(* Logix 5000 project; controller AdvManLab vendor 1 type 14 code 158 rev 28.12; software revision 28.01; part 3 of 13 *)
(* tags used below, declared in another part *)
   Cfg_Exists : BOOL;   // 1=Alarm configured to exist, 0=Does not exist, don't scan
   Cfg_ResetReqd : BOOL;   // 1=Latched Alarm, a Reset is required to clear this Alarm
   Cfg_AckReqd : BOOL;   // 1=Acknowledge required for this Alarm
   Cfg_AllowShelve : BOOL;   // 1=Allow Operator to Shelve this Alarm
   Cfg_AllowDisable : BOOL;   // 1=Allow Maintenance to Disable this Alarm
   Cfg_Severity : INT;   // Alarm Severity: 1..250=Low, 251..500=Medium, 501..750=High, 751..1000=Urgent
   Cfg_AlmMinOnT : DINT;   // Minimum time Alm output stays on (sec)
   PCfg_AllowExist : BOOL;   // 1=Alarm can be configured to exist, 0=other configs make alarm meaningless
   PCmd_Ack : BOOL;   // Program Command to Acknowledge alarm
   PCmd_Suppress : BOOL;   // Program Command to Suppress by Design (inhibits new alarm)
   PCmd_Unsuppress : BOOL;   // Program Command to Unsuppress (allows new alarm)
   PCmd_Unshelve : BOOL;   // Program Command to Unshelve (e.g., on shift change)
   OCmd_Ack : BOOL;   // Operator Command to Acknowledge alarm
   OCmd_Shelve : BOOL;   // Operator Command to Shelve Alarm (inhibits new alarm)
   OCmd_Unshelve : BOOL;   // Operator Command to Unshelve alarm (allows new alarm)
   Alm : ALIAS FOR Com_AE.0;   // Alarm output 1=In Alarm
   Ack : ALIAS FOR Com_AE.1;   // Alarm acknowledged status: 1=Ack rcvd
   Shelved : ALIAS FOR Com_AE.3;   // 1=Alarm has been Shelved by Operator (inhibits new alarm)
   Suppressed : ALIAS FOR Com_AE.6;   // 1=Alarm has been Suppressed by Program (inhibits new alarm)
   Disabled : ALIAS FOR Com_AE.9;   // 1=Alarm has been Disabled by Maintanance (inhibits new alarm)
   P_Alarm : BOOL;   // Unique Parameter Name for auto - discovery
   Wrk_Suppressed : BOOL;   // Internal Alarm Suppressed Status
   Com_AE : INT;   // Communication with HMI / Alarm/Event Server (see bit descriptions)
   PF525 : PF525_Faceplate_AOI;
   Running : BOOL;
(* P_Alarm, continued *)

ROUTINE Prescan   (* ladder *)
// Clear "lurking" Commands
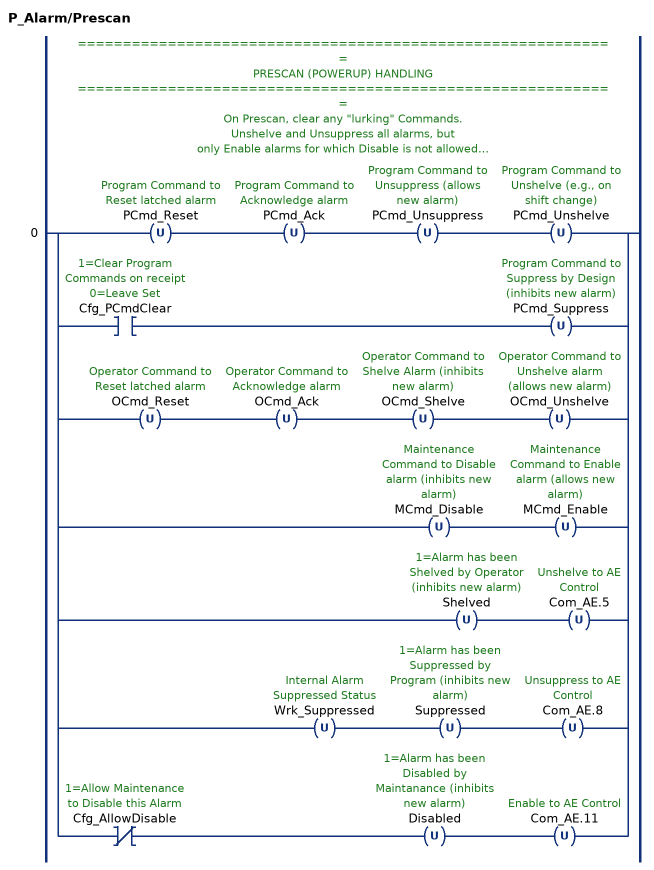
   // ============================================================
   // PRESCAN (POWERUP) HANDLING
   // ============================================================
   // On Prescan, clear any "lurking" Commands.
   // Unshelve and Unsuppress all alarms, but
   // only Enable alarms for which Disable is not allowed.
   // (Let Maintenance Disable persist through a power cycle...)
   // #####  V3.0-00  2013-06-30:  Added PCmd_Unshelve, AllowDisable, AllowShelve.  #####
   0: [OTU(PCmd_Reset) OTU(PCmd_Ack) OTU(PCmd_Unsuppress) OTU(PCmd_Unshelve) ,XIC(Cfg_PCmdClear) OTU(PCmd_Suppress) ,OTU(OCmd_Reset) OTU(OCmd_Ack) OTU(OCmd_Shelve) OTU(OCmd_Unshelve) ,OTU(MCmd_Disable) OTU(MCmd_Enable) ,OTU(Shelved) OTU(Com_AE.5) ,OTU(Wrk_Suppressed) OTU(Suppressed) OTU(Com_AE.8) ,XIO(Cfg_AllowDisable) OTU(Disabled) OTU(Com_AE.11) ];
END_ROUTINE
END_ADD_ON_INSTRUCTION

ADD_ON_INSTRUCTION P_Mode   (* revision 3.1 00 Release, vendor Rockwell Automation, ExecutePrescan, ExecuteEnableInFalse *)
// Mode
// Revision note:
// See Release Notes for Library version 3.1-xx for details. Containing objects must expose Maintenance
// Acquire / Release commands and new Sts_MAcqRcvd.
// Changed Val (enum) to SINT. Fixed parameter descriptions.
// Help:
// Copyright © Rockwell Automation, Inc.  All Rights Reserved.
// This instruction provides selection of Mode (owner) for a Device level
// object  (from highest priority to lowest):
// *  No Mode (no owner, EnableIn is false)
// *  Hand (typically tracks hardwired control of device)
// *  Maint (Maintenance) (taken out of normal service for maintenance)
// *  Ovrd (Override) (typically used for process overrides)
// *  Prog  (Program) (automated control, and default if Cfg_ProgNorm = 1)
// *  Oper (Operator (manual control, and default if Cfg_ProgNorm = 0)
// (Program and Operator have the same priority.)
// The current mode is shown with Status bits and also as the primary
// Value for the instruction: an enumeration "Val" as follows:
//   0 = No Mode,
//   1 = Hand,
//   2 = Maintenance,
//   3 = Override,
//   4 = Program (Locked),
//   5 = Operator (Locked),
//   6 = Program (Unlocked, Oper default),
//   7 = Operator (Unlocked, Prog default),
//   8 = Program (Unlocked, = default),
//   9 = Operator (Unlocked, = default).
// When EnableIn is false, all ownership acquire/release and lock/unlock
// Commands are processed "behind the scenes", but the Mode is shown
// as "No Mode" (no owner).  When EnableIn becomes true, the Mode
// takes into account the Commands received -- in other words, the Mode
// becomes the one that would have been in effect had the EnableIn
// False / No Mode condition never occurred.
VAR_INPUT
   Inp_Hand : BOOL; {visible}   // 1=Acquire Hand (typ. hardwired local) Mode, 0=Release Hand Mode
   Inp_Ovrd : BOOL; {visible}   // 1=Acquire Override (higher priority program logic) Mode, 0=Release Override Mode
   Cfg_PCmdClear : BOOL := 1;   // 1=Clear Program Command on receipt; 0=Use Level-based (maintained) PCmds
   Cfg_OvrdOverLock : BOOL := 1;   // 1=Override supersedes Prog/Oper Lock, 0=don't override Lock
   Cfg_ProgDefault : BOOL;   // Default Mode: 1=Program Mode if no requests; 0=Operator Mode if no requests
   PCmd_Acq : BOOL;   // Program Command to Acquire Ownership (Oper to Prog)
   PCmd_Rel : BOOL;   // Program Command to Release Ownership (Prog to Oper)
   PCmd_Lock : BOOL;   // Program Command to Lock Mode in Prog
   PCmd_Unlock : BOOL;   // Program Command to Unlock Mode
   MCmd_Acq : BOOL;   // Maintenance Command to Acquire Ownership (Oper/Prog/Ovrd to Maint)
   MCmd_Rel : BOOL;   // Maintenance Command to Release Ownership (Maint to Oper/Prog/Ovrd)
   OCmd_AcqLock : BOOL;   // Operator Command to Acquire (Prog to Oper) / Lock Ownership
   OCmd_UnlockRel : BOOL;   // Operator Command to Unlock / Release (Oper to Prog) Ownership
END_VAR
VAR_OUTPUT
   Val : SINT; {access Read Only}   // Mode enum: 0=No, 1=H, 2=M, 3=!, 4=P Lock, 5=O Lock, 6=P (O Def), 7=O (P Def), 8=P (= Def), 9=O (= Def)
   Sts_Hand : BOOL; {access Read Only, visible}   // 1=Mode is Hand (supersedes Maint, Ovrd, Prog, Oper)
   Sts_Maint : BOOL; {access Read Only, visible}   // 1=Mode is Maintenance (supersedes Ovrd, Prog, Oper)
   Sts_Ovrd : BOOL; {access Read Only, visible}   // 1=Mode is Override (supersedes Prog, Oper)
   Sts_Prog : BOOL; {access Read Only, visible}   // 1=Mode is Program
   Sts_Oper : BOOL := 1; {access Read Only, visible}   // 1=Mode is Operator
   Sts_ProgOperLock : BOOL; {access Read Only, visible}   // 1=Program or Operator has requested Mode Lock
   Sts_ProgOperSel : BOOL; {access Read Only}   // Prog/Oper selection 1=Program, 0=Operator
   Sts_NoMode : BOOL; {access Read Only}   // 1=Mode is No Mode (no owner, disabled or not scanned)
   Sts_MAcqRcvd : BOOL; {access Read Only}   // 1=Maintenance Acquire command received this scan
   Rdy_MAcq : BOOL; {access Read Only}   // 1=Ready for MCmd_Acq, enable button
   Rdy_MRel : BOOL; {access Read Only}   // 1=Ready for MCmd_Rel, enable button
   Rdy_OAcq : BOOL; {access Read Only}   // 1=Ready for OCmd_AcqLock, enable Acquire (to Oper) button
   Rdy_OLock : BOOL; {access Read Only}   // 1=Ready for OCmd_AcqLock, enable Oper Lock button
   Rdy_OUnlock : BOOL; {access Read Only}   // 1=Ready for OCmd_UnlockRel, enable Oper Unlock button
   Rdy_ORel : BOOL; {access Read Only}   // 1=Ready for OCmd_UnlockRel, enable Release (to Prog) button
   P_Mode : BOOL;   // Unique Parameter Name for auto - discovery
END_VAR
VAR
   Wrk_Locked : BOOL; {access None}   // 1=Program/Operator Mode selection is Locked
   Wrk_Prog : BOOL; {access None}   // Internal Program (1) / Operator (0) Mode selection
   Wrk_Maint : BOOL; {access None}   // Internal Maintenance Mode
   Inf_Lib : STRING_12 := 'RA-BAS'; {access Read Only}   // Display Library for Faceplate call-up
   Inf_Type : STRING_16 := 'P_Mode'; {access Read Only}   // Must contain AOI name, used for HMI and Information S/W
END_VAR

ROUTINE EnableInFalse   (* ladder *)
// Processes received Commands, but shows "NO mode" (no owner)
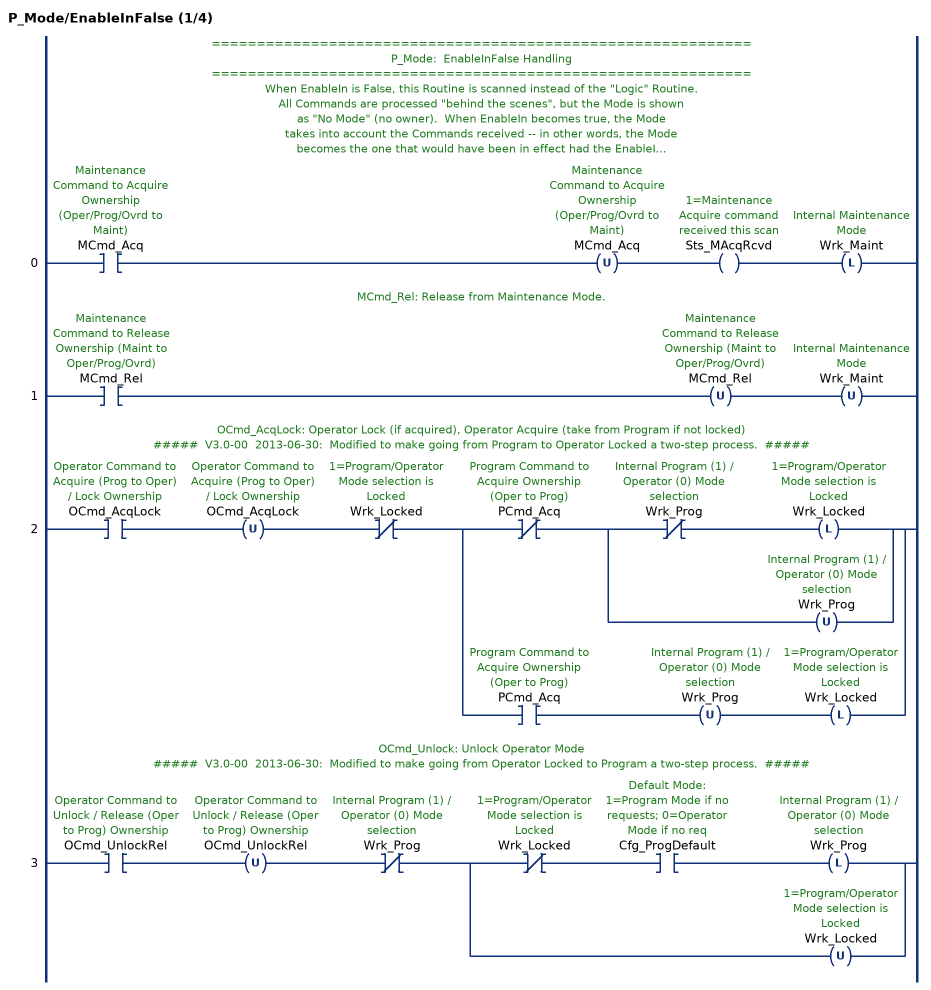
   // ============================================================
   // P_Mode:  EnableInFalse Handling
   // ============================================================
   // When EnableIn is False, this Routine is scanned instead of the "Logic" Routine.
   // All Commands are processed "behind the scenes", but the Mode is shown
   // as "No Mode" (no owner).  When EnableIn becomes true, the Mode
   // takes into account the Commands received -- in other words, the Mode
   // becomes the one that would have been in effect had the EnableIn
   // False / No Mode condition never occurred.
   // ============================================================
   // COMMAND HANDLING
   // ============================================================
   // NOTE:  These rungs MUST be in the order given to meet the following
   // multiple-actions-at-the-same-time scenarios:
   // * Maintenance Release beats Maintenance Acquire
   // * Program Release beats Program Acquire
   // * Program Unlock beats Program Lock
   // * Operator Unlock beats Operator Acquire and Lock (results in Oper Unlocked)
   // * Operator Acquire/Lock must come after Program Unlock
   // * Program Acquire must come after Operator Unlock
   // ===========================================================
   // MCmd_Acq: Acquire for Maintenance Mode, and blink the status
   // that indicates a Maintenance Acquire command was received.
   // #####  V3.1-00  2014-06-30:  Added Sts_MAcqRcvd  #####
   0: XIC(MCmd_Acq)OTU(MCmd_Acq)OTE(Sts_MAcqRcvd)OTL(Wrk_Maint);
   // MCmd_Rel: Release from Maintenance Mode.
   1: XIC(MCmd_Rel)OTU(MCmd_Rel)OTU(Wrk_Maint);
   // OCmd_AcqLock: Operator Lock (if acquired), Operator Acquire (take from Program if not locked)
   // #####  V3.0-00  2013-06-30:  Modified to make going from Program to Operator Locked a two-step process.  #####
   2: XIC(OCmd_AcqLock)OTU(OCmd_AcqLock)XIO(Wrk_Locked)[XIO(PCmd_Acq) [XIO(Wrk_Prog) OTL(Wrk_Locked) ,OTU(Wrk_Prog) ] ,XIC(PCmd_Acq) OTU(Wrk_Prog) OTL(Wrk_Locked) ];
   // OCmd_Unlock: Unlock Operator Mode
   // #####  V3.0-00  2013-06-30:  Modified to make going from Operator Locked to Program a two-step process.  #####
   3: XIC(OCmd_UnlockRel)OTU(OCmd_UnlockRel)XIO(Wrk_Prog)[XIO(Wrk_Locked) XIC(Cfg_ProgDefault) OTL(Wrk_Prog) ,OTU(Wrk_Locked) ];
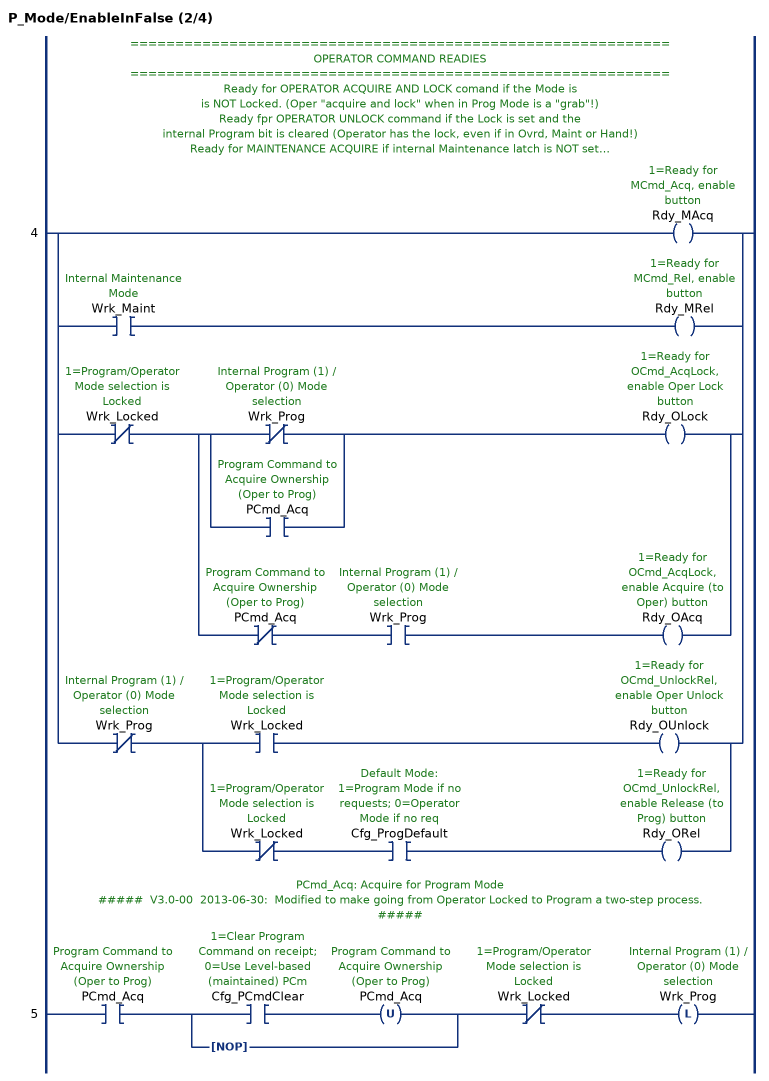
   // ============================================================
   // OPERATOR COMMAND READIES
   // ============================================================
   // Ready for OPERATOR ACQUIRE AND LOCK comand if the Mode is
   //  is NOT Locked. (Oper "acquire and lock" when in Prog Mode is a "grab"!)
   // Ready fpr OPERATOR UNLOCK command if the Lock is set and the
   // internal Program bit is cleared (Operator has the lock, even if in Ovrd, Maint or Hand!)
   // Ready for MAINTENANCE ACQUIRE if internal Maintenance latch is NOT set.
   // But we need to display Ready even if latch IS set so that Sts_MAcqRcvd
   // can blink to reset an external Maintenance expiration timer!!!
   // Ready for MAINTENANCE RELEASE if internal Maintenance latch IS set.
   // #####  V3.0-00  2013-06-30:  Modified Rdy_Unlock for two-step Operator Locked to Program process.  #####
   // #####  V3.1-00  2014-06-30:  Added Sts_MAcqRcvd  #####
   4: [OTE(Rdy_MAcq) ,XIC(Wrk_Maint) OTE(Rdy_MRel) ,XIO(Wrk_Locked) [[XIO(Wrk_Prog) ,XIC(PCmd_Acq) ] OTE(Rdy_OLock) ,XIO(PCmd_Acq) XIC(Wrk_Prog) OTE(Rdy_OAcq) ] ,XIO(Wrk_Prog) [XIC(Wrk_Locked) OTE(Rdy_OUnlock) ,XIO(Wrk_Locked) XIC(Cfg_ProgDefault) OTE(Rdy_ORel) ] ];
   // PCmd_Acq: Acquire for Program Mode
   // #####  V3.0-00  2013-06-30:  Modified to make going from Operator Locked to Program a two-step process.  #####
   5: XIC(PCmd_Acq)[XIC(Cfg_PCmdClear) OTU(PCmd_Acq) ,NOP() ]XIO(Wrk_Locked)OTL(Wrk_Prog);
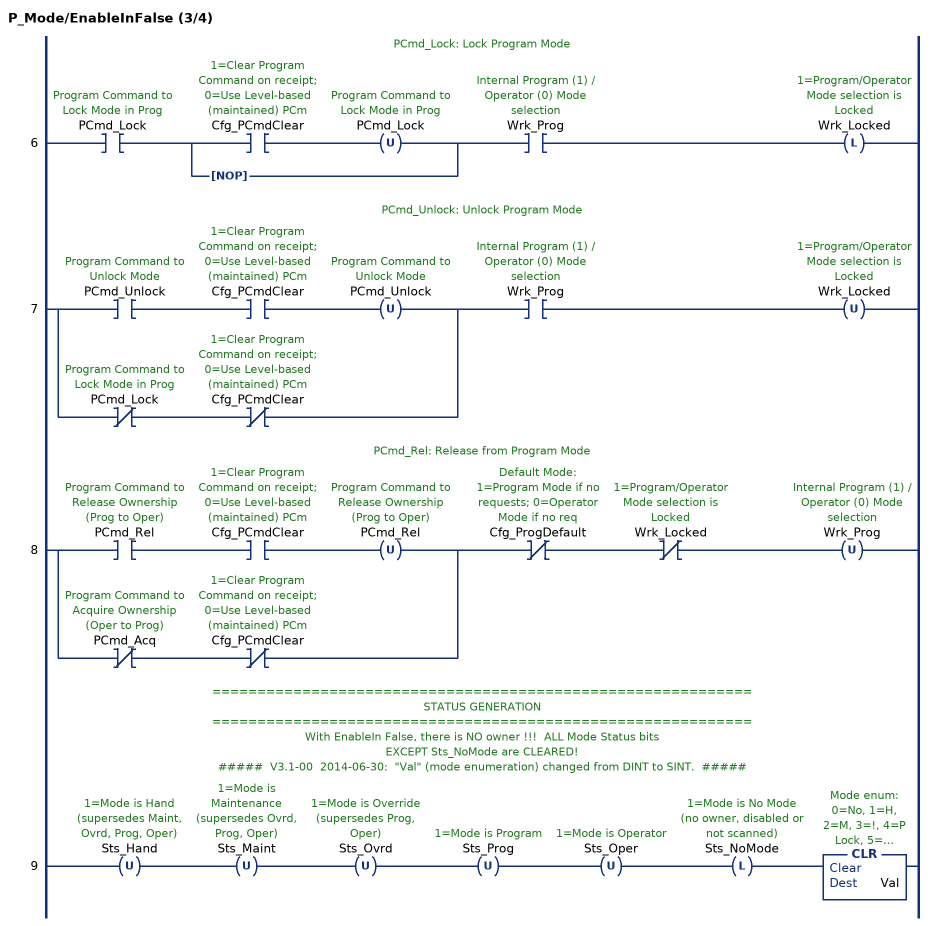
   // PCmd_Lock: Lock Program Mode
   6: XIC(PCmd_Lock)[XIC(Cfg_PCmdClear) OTU(PCmd_Lock) ,NOP() ]XIC(Wrk_Prog)OTL(Wrk_Locked);
   // PCmd_Unlock: Unlock Program Mode
   7: [XIC(PCmd_Unlock) XIC(Cfg_PCmdClear) OTU(PCmd_Unlock) ,XIO(PCmd_Lock) XIO(Cfg_PCmdClear) ]XIC(Wrk_Prog)OTU(Wrk_Locked);
   // PCmd_Rel: Release from Program Mode
   8: [XIC(PCmd_Rel) XIC(Cfg_PCmdClear) OTU(PCmd_Rel) ,XIO(PCmd_Acq) XIO(Cfg_PCmdClear) ]XIO(Cfg_ProgDefault)XIO(Wrk_Locked)OTU(Wrk_Prog);
   // ============================================================
   // STATUS GENERATION
   // ============================================================
   // With EnableIn False, there is NO owner !!!  ALL Mode Status bits
   // EXCEPT Sts_NoMode are CLEARED!
   // #####  V3.1-00  2014-06-30:  "Val" (mode enumeration) changed from DINT to SINT.  #####
   9: OTU(Sts_Hand)OTU(Sts_Maint)OTU(Sts_Ovrd)OTU(Sts_Prog)OTU(Sts_Oper)OTL(Sts_NoMode)CLR(Val);
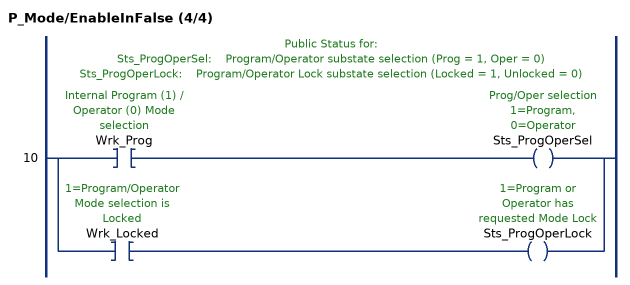
   // Public Status for:
   // Sts_ProgOperSel:    Program/Operator substate selection (Prog = 1, Oper = 0)
   // Sts_ProgOperLock:    Program/Operator Lock substate selection (Locked = 1, Unlocked = 0)
   10: [XIC(Wrk_Prog) OTE(Sts_ProgOperSel) ,XIC(Wrk_Locked) OTE(Sts_ProgOperLock) ];
END_ROUTINE

ROUTINE Logic   (* ladder *)
// Selects Modes (Hand, Maint, Ovrd, Oper, Prog) based on Inputs and Commands
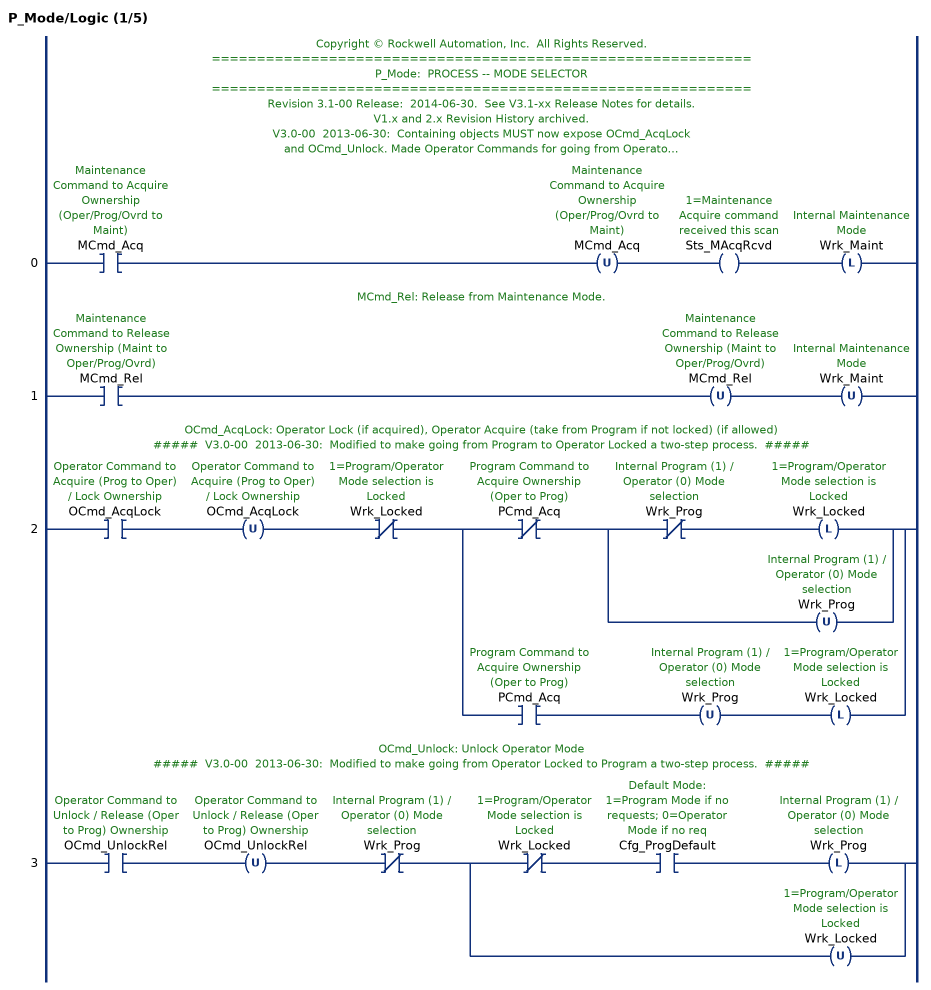
   // Copyright © Rockwell Automation, Inc.  All Rights Reserved.
   // ============================================================
   // P_Mode:  PROCESS -- MODE SELECTOR
   // ============================================================
   // Revision 3.1-00 Release:  2014-06-30.  See V3.1-xx Release Notes for details.
   // V1.x and 2.x Revision History archived.
   // V3.0-00  2013-06-30:  Containing objects MUST now expose OCmd_AcqLock
   // and OCmd_Unlock. Made Operator Commands for going from Operator
   // Locked to Program (unlocked) and Program (unlocked) to Operator
   // Lock two-step processes.  Added Inf_Lib, Inf_Type.
   // V3.1-00  2014-06-30: Containing objects must expose Maintenance
   // Acquire / Release commands and new Sts_MAcqRcvd.
   // Changed Val (enum) to SINT. Fixed parameter descriptions.
   // ============================================================
   // This instruction provides selection of Mode (owner) for a Device level
   // object  (from highest priority to lowest):
   // * NO Mode (EnableIn is false)
   // *  Hand (typically tracks hardwired control of device)
   // *  Maint (Maintenance) (taken out of normal service for maintenance)
   // *  Ovrd (Override) (typically used for process overrides)
   // *  Prog  (Program) (automated control, and default if Cfg_ProgNorm = 1)
   // *  Oper (Operator (manual control, and default if Cfg_ProgNorm = 0)
   // The current mode is shown with Status bits and also as the
   // primary Value for the instruction: an enumeration as follows:
   // 0 = No Mode, 1 = Hand, 2 = Maintenance, 3 = Override,
   // 4 = Program (Locked), 5 = Operator (Locked),
   // 6 = Program (Unlocked, Oper default), 7 = Operator (Unlocked, Prog default),
   // 8 = Program (Unlocked, Prog default), 9 = Operator (Unlocked, Oper default).
   // ============================================================
   // COMMAND HANDLING
   // ============================================================
   // NOTE:  These rungs MUST be in the order given to meet the following
   // multiple-actions-at-the-same-time scenarios:
   // * Maintenance Release beats Maintenance Acquire
   // * Program Release beats Program Acquire
   // * Program Unlock beats Program Lock
   // * Operator Unlock beats Operator Acquire / Lock (results in Oper Unlocked)
   // * Program Acquire must come after Operator Unlock
   // If Cfg_ProgDefault = 1, the Mode defaults to Program
   // (instead of Operator) if all other Modes release their requests.
   // ============================================================
   // MCmd_Acq: Acquire for Maintenance Mode, and blink the status
   // that indicates a Maintenance Acquire command was received.
   // #####  V3.1-00  2014-06-30:  Added Sts_MAcqRcvd  #####
   0: XIC(MCmd_Acq)OTU(MCmd_Acq)OTE(Sts_MAcqRcvd)OTL(Wrk_Maint);
   // MCmd_Rel: Release from Maintenance Mode.
   1: XIC(MCmd_Rel)OTU(MCmd_Rel)OTU(Wrk_Maint);
   // OCmd_AcqLock: Operator Lock (if acquired), Operator Acquire (take from Program if not locked) (if allowed)
   // #####  V3.0-00  2013-06-30:  Modified to make going from Program to Operator Locked a two-step process.  #####
   2: XIC(OCmd_AcqLock)OTU(OCmd_AcqLock)XIO(Wrk_Locked)[XIO(PCmd_Acq) [XIO(Wrk_Prog) OTL(Wrk_Locked) ,OTU(Wrk_Prog) ] ,XIC(PCmd_Acq) OTU(Wrk_Prog) OTL(Wrk_Locked) ];
   // OCmd_Unlock: Unlock Operator Mode
   // #####  V3.0-00  2013-06-30:  Modified to make going from Operator Locked to Program a two-step process.  #####
   3: XIC(OCmd_UnlockRel)OTU(OCmd_UnlockRel)XIO(Wrk_Prog)[XIO(Wrk_Locked) XIC(Cfg_ProgDefault) OTL(Wrk_Prog) ,OTU(Wrk_Locked) ];
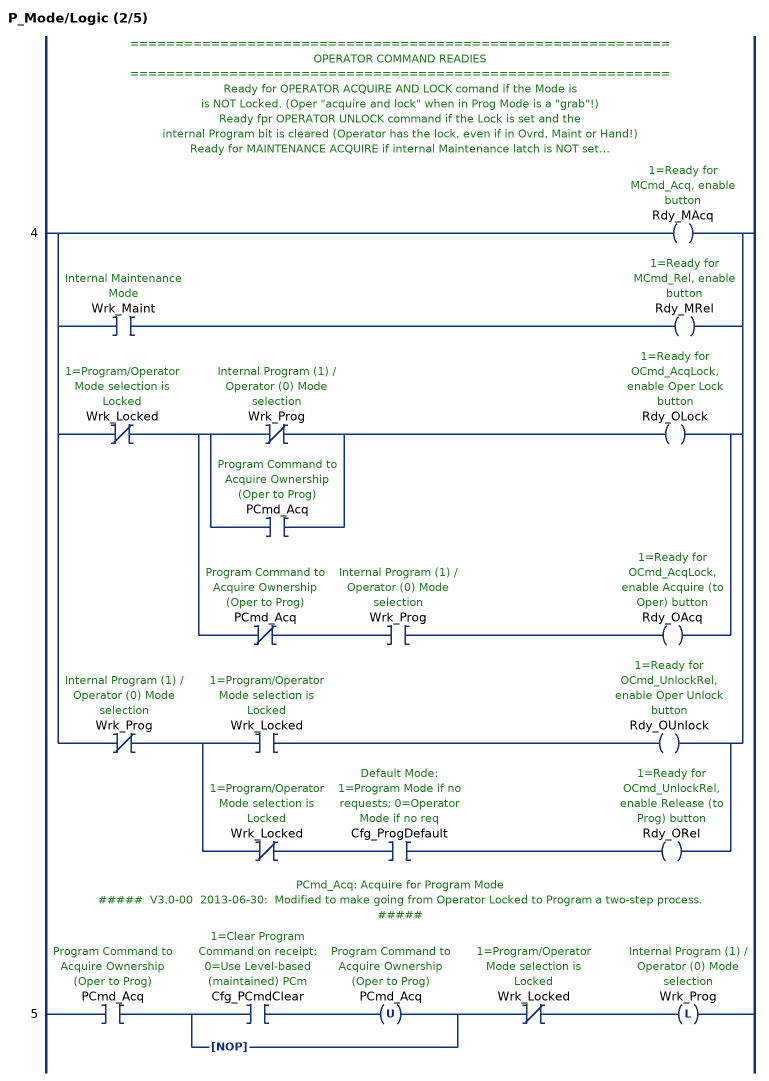
   // ============================================================
   // OPERATOR COMMAND READIES
   // ============================================================
   // Ready for OPERATOR ACQUIRE AND LOCK comand if the Mode is
   //  is NOT Locked. (Oper "acquire and lock" when in Prog Mode is a "grab"!)
   // Ready fpr OPERATOR UNLOCK command if the Lock is set and the
   // internal Program bit is cleared (Operator has the lock, even if in Ovrd, Maint or Hand!)
   // Ready for MAINTENANCE ACQUIRE if internal Maintenance latch is NOT set.
   // But we need to display Ready even if latch IS set so that Sts_MAcqRcvd
   // can blink to reset an external Maintenance expiration timer!!!
   // Ready for MAINTENANCE RELEASE if internal Maintenance latch IS set.
   // #####  V3.0-00  2013-06-30:  Modified Rdy_Unlock for two-step Operator Locked to Program process.  #####
   // #####  V3.1-00  2014-06-30:  Added Sts_MAcqRcvd  #####
   4: [OTE(Rdy_MAcq) ,XIC(Wrk_Maint) OTE(Rdy_MRel) ,XIO(Wrk_Locked) [[XIO(Wrk_Prog) ,XIC(PCmd_Acq) ] OTE(Rdy_OLock) ,XIO(PCmd_Acq) XIC(Wrk_Prog) OTE(Rdy_OAcq) ] ,XIO(Wrk_Prog) [XIC(Wrk_Locked) OTE(Rdy_OUnlock) ,XIO(Wrk_Locked) XIC(Cfg_ProgDefault) OTE(Rdy_ORel) ] ];
   // PCmd_Acq: Acquire for Program Mode
   // #####  V3.0-00  2013-06-30:  Modified to make going from Operator Locked to Program a two-step process.  #####
   5: XIC(PCmd_Acq)[XIC(Cfg_PCmdClear) OTU(PCmd_Acq) ,NOP() ]XIO(Wrk_Locked)OTL(Wrk_Prog);
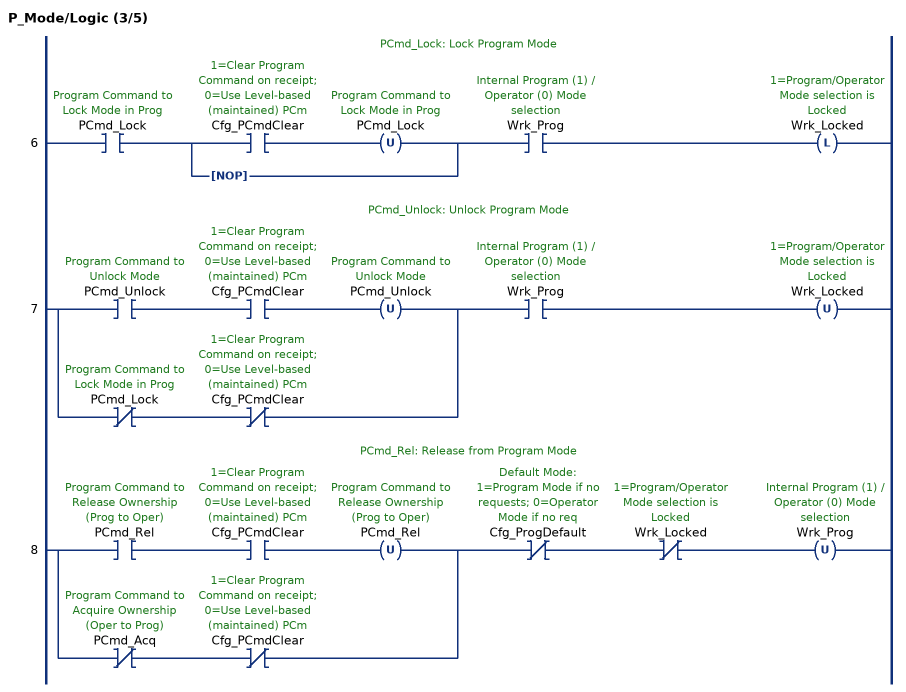
   // PCmd_Lock: Lock Program Mode
   6: XIC(PCmd_Lock)[XIC(Cfg_PCmdClear) OTU(PCmd_Lock) ,NOP() ]XIC(Wrk_Prog)OTL(Wrk_Locked);
   // PCmd_Unlock: Unlock Program Mode
   7: [XIC(PCmd_Unlock) XIC(Cfg_PCmdClear) OTU(PCmd_Unlock) ,XIO(PCmd_Lock) XIO(Cfg_PCmdClear) ]XIC(Wrk_Prog)OTU(Wrk_Locked);
   // PCmd_Rel: Release from Program Mode
   8: [XIC(PCmd_Rel) XIC(Cfg_PCmdClear) OTU(PCmd_Rel) ,XIO(PCmd_Acq) XIO(Cfg_PCmdClear) ]XIO(Cfg_ProgDefault)XIO(Wrk_Locked)OTU(Wrk_Prog);
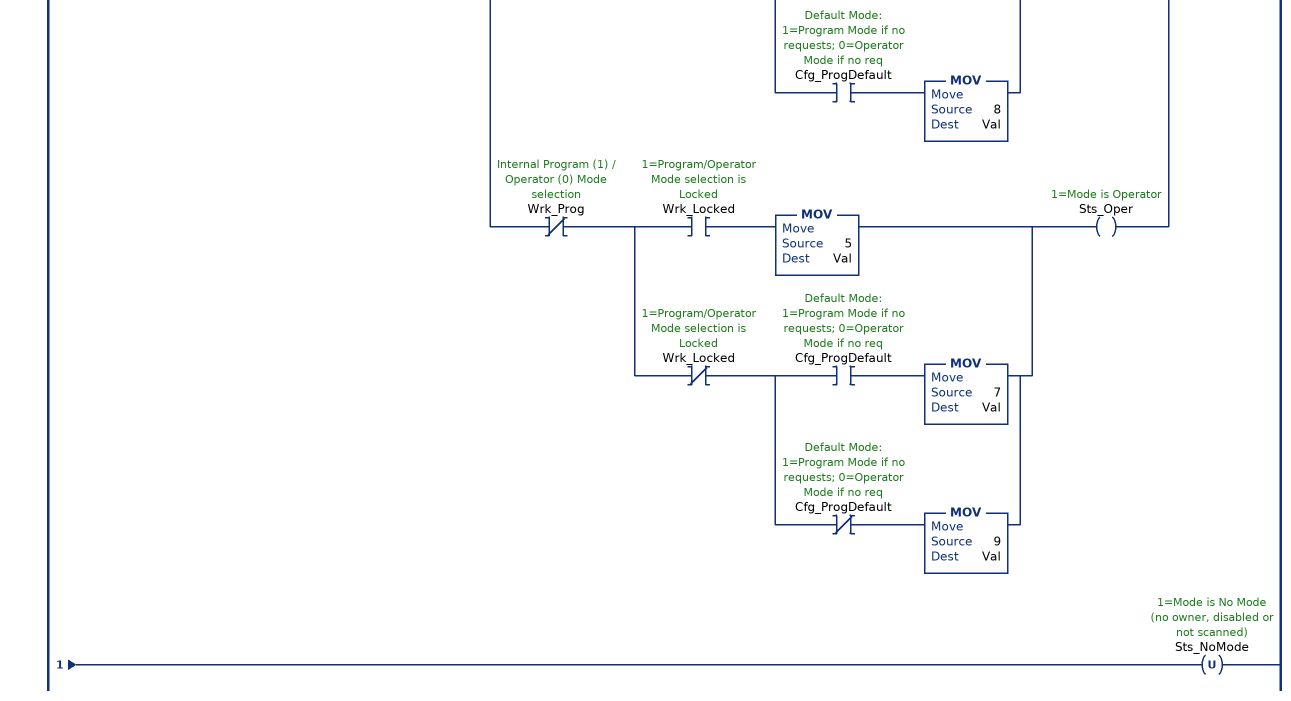
   // ============================================================
   // STATUS GENERATION
   // ============================================================
   // This rung determines the Mode based on the states of the inputs and internal working bits.
   // The logic here does the vast mahority of the implementation of the Mode selection rules.
   // Between the internal working bits used above and the rules implemented here,
   // outside objects cannot manipulate the state of this object by setting/clearing its Status bits.
   // Public Status is generated for:
   // *  Hand Mode
   // *  Maintenance Mode
   // *  Override Mode
   // *  Program Mode
   // *  Operator Mode
   // *  No Mode (none of the above)
   // #####  V3.1-00  2014-06-30:  "Val" (mode enumeration) changed from DINT to SINT.  #####
   9: [XIC(Inp_Hand) OTE(Sts_Hand) MOV(1,Val) ,XIO(Inp_Hand) [XIC(Wrk_Maint) OTE(Sts_Maint) MOV(2,Val) ,XIO(Wrk_Maint) [XIC(Inp_Ovrd) [XIO(Wrk_Locked) ,XIC(Cfg_OvrdOverLock) ,XIC(Sts_Ovrd) ] OTE(Sts_Ovrd) MOV(3,Val) ,XIO(Sts_Ovrd) [XIC(Wrk_Prog) [XIC(Wrk_Locked) MOV(4,Val) ,XIO(Wrk_Locked) [XIO(Cfg_ProgDefault) MOV(6,Val) ,XIC(Cfg_ProgDefault) MOV(8,Val) ] ] OTE(Sts_Prog) ,XIO(Wrk_Prog) [XIC(Wrk_Locked) MOV(5,Val) ,XIO(Wrk_Locked) [XIC(Cfg_ProgDefault) MOV(7,Val) ,XIO(Cfg_ProgDefault) MOV(9,Val) ] ] OTE(Sts_Oper) ] ] ] ]OTU(Sts_NoMode);
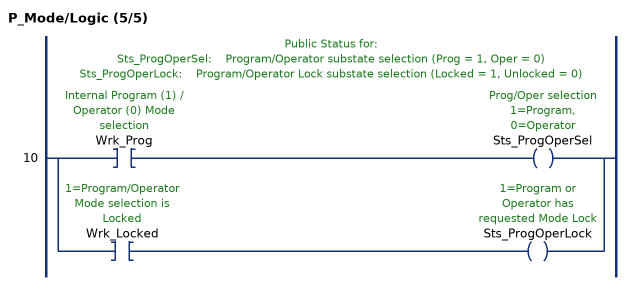
   // Public Status for:
   // Sts_ProgOperSel:    Program/Operator substate selection (Prog = 1, Oper = 0)
   // Sts_ProgOperLock:    Program/Operator Lock substate selection (Locked = 1, Unlocked = 0)
   10: [XIC(Wrk_Prog) OTE(Sts_ProgOperSel) ,XIC(Wrk_Locked) OTE(Sts_ProgOperLock) ];
END_ROUTINE

ROUTINE Prescan   (* ladder *)
// Clear "lurking" Commands
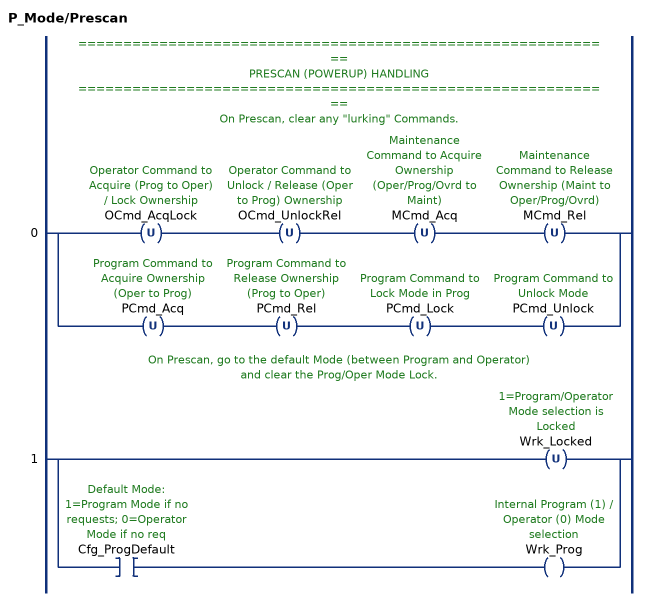
   // ============================================================
   // PRESCAN (POWERUP) HANDLING
   // ============================================================
   // On Prescan, clear any "lurking" Commands.
   0: [OTU(OCmd_AcqLock) OTU(OCmd_UnlockRel) OTU(MCmd_Acq) OTU(MCmd_Rel) ,OTU(PCmd_Acq) OTU(PCmd_Rel) OTU(PCmd_Lock) OTU(PCmd_Unlock) ];
   // On Prescan, go to the default Mode (between Program and Operator)
   // and clear the Prog/Oper Mode Lock.
   1: [OTU(Wrk_Locked) ,XIC(Cfg_ProgDefault) OTE(Wrk_Prog) ];
END_ROUTINE
END_ADD_ON_INSTRUCTION

ADD_ON_INSTRUCTION P_PF52x   (* revision 3.1 00 Release, vendor Rockwell Automation, ExecutePrescan, ExecuteEnableInFalse *)
// PowerFlex 523 / 525
// Variable Frequency Drive
// Revision note:
// See V3.1-xx Release Notes for Library for details. New instruction for PlantPAx Library 3.1.
// Help:
// Copyright © Rockwell Automation, Inc.  All Rights Reserved.
// This Instruction controls and monitors a PowerFlex 523 Variable-Frequency Drive with
// optional EtherNet/IP Interface, or a PowerFlex 525 Variable-Frequency Drive with
// embedded or optional add-on EtherNet/IP Interface.
// This instruction provides:
// *  Starting, stopping, jogging of drive, setting speed reference and direction
// *  Monitoring of run feedback, display of actual drive status, including accel, decel, direction, speed
// *  Detection of Failure to Start, Failure to Stop, Drive Fault
// *  Monitoring of Permissive conditions to allow starting
// *  Monitoring of Interlock conditions to stop / prevent starting
// *  Simulation, providing feedback of a working drive while disabling outputs
// *  Monitoring of I/O communication faults
// *  Alarms for Fail to Start, Fail to Stop, Interlock Trip, Drive Fault, I/O Fault
// *  Option to automatically reset faults and alarms when operator commands
//     motor to start or stop
// * Supports HMI "breadcrumbs" for Alarm Inhibited, Bad Configuration,
//     Not Ready, Maintenance Bypass Active
// * "Available" status for use by automation logic to know whether motor
//     can be controlled by other objects.
// See Rockwell Automation Publication 520COM-UM001_ for information on
// the PowerFlex 525 embedded EtherNet/IP interface.
// See Rockwell Automation Publication 520COM-UM003_ for information on
// the PowerFlex 525 add-on EtherNet/IP interface (dual-port).
// See Rockwell Automation Publication 520-UM001_ for information on the
// PowerFlex 523 and 525 drive parameters and programming
// Modes are provided by a P_Mode AOI instance.
// Alarms are provided by P_Alarm AOI instances.
// Modes of operation: Operator, Program, Override, Maintenance, Hand
// REQUIRED DRIVE CONFIGURATION
// Be certain to set up the drive Datalinks as follows!
// 'User Choice' Datalinks are not used by this AOI and
// may be left unused or set up for your application.
// INPUT ASSEMBLY:
// Drive Status (standard)
// Output Frequency (standard)
// 1. Fault 1 Code (Par 007)
// 2. Output Current (Par 003)
// 3. Output Power (Par 017)
// 4. User choice
// OUTPUT ASSEMBLY:
// Drive Logic Comnmand (standard)
// Frequency Command (Speed Reference) (standard)
// All 4 output datalinks are user choice.
VAR_IN_OUT
   Inp : P_PF52x_Inp; {required}   // Common part of PF523 / PF525 Input Assembly
   Out : P_PF52x_Out; {required}   // Common part of PF523 / PF525 Output Assembly
   Ref_FaultCodeList : P_DescList[1]; {required}   // Tag containing List of Fault Codes (DINT) and their Descriptions (STRING)
END_VAR
VAR_INPUT
   Inp_FwdPermOK : BOOL := 1; {visible}   // 1=Permissives OK, drive can start Forward
   Inp_FwdNBPermOK : BOOL := 1; {visible}   // 1=Non-Bypassable Permissives OK, drive can start Forward
   Inp_RevPermOK : BOOL := 1; {visible}   // 1=Permissives OK, drive can start Reverse
   Inp_RevNBPermOK : BOOL := 1; {visible}   // 1=Non-Bypassable Permissives OK, motor can start Reverse
   Inp_IntlkOK : BOOL := 1; {visible}   // 1=Interlocks OK, drive can start/run
   Inp_NBIntlkOK : BOOL := 1; {visible}   // 1=Non-Bypassable Interlocks OK, drive can start/run
   Inp_IOFault : BOOL;   // Input Communication Status 0=OK, 1=fail
   Inp_Sim : BOOL;   // 1=Simulate working drive; 0=Start/Stop/ Monitor actual drive
   Inp_Hand : BOOL; {visible}   // 1=Acquire Hand (typ. hardwired local) Mode, 0=Release Hand Mode
   Inp_Ovrd : ALIAS FOR Mode.Inp_Ovrd; {visible}
   Inp_OvrdCmd : SINT; {visible}   // Override Mode Command: 0=None, 1=Stop, 2=Start Fwd 3=Start Rev
   Inp_OvrdSpeed : REAL;   // Value to set Speed Reference in Override Mode (SpeedRef EU)
   Inp_Reset : BOOL; {visible}   // 1=Reset drive fault conditions and latched Alarms
   Cfg_HasReverse : BOOL;   // 1=Drive can be run reverse, 0=Forward only
   Cfg_HasJog : BOOL;   // 1=Drive Jog Command enabled/visible, 0=Drive Jog Command not allowed
   Cfg_AllowLocal : BOOL;   // 1=Allow Local Start/Stop without alarm, 0=Start/Stop from HMI/prog only
   Cfg_HasFwdPermObj : BOOL;   // 1=Tells HMI a P_Perm is connected to Inp_FwdPerm
   Cfg_HasRevPermObj : BOOL;   // 1=Tells HMI a P_Perm is connected to Inp_RevPerm
   Cfg_HasIntlkObj : BOOL;   // 1=Tells HMI a P_Intlk is connected to Inp_Intlk
   Cfg_HasResInhObj : BOOL;   // 1=Tells HMI a P_ResInh Restart Inhibit is connected
   Cfg_HasRunTimeObj : BOOL;   // 1=Tells HMI a P_RunTime is connected
   Cfg_SetTrack : BOOL := 1;   // 1=PSets track OSets in Oper, OSets track PSets in Prog, 0=no tracking
   Cfg_SetTrackOvrdHand : BOOL;   // 1=Prog/Oper Settings track Override/Hand speed reference
   Cfg_PCmdClear : ALIAS FOR Mode.Cfg_PCmdClear;
   Cfg_ProgDefault : ALIAS FOR Mode.Cfg_ProgDefault;
   Cfg_OperStopPrio : BOOL;   // 1=OCmd_Stop has priority, accepted any time, 0=OCmd_Stop only in Oper, Maint Mode.
   Cfg_OCmdResets : BOOL;   // 1=New Oper drive cmd. resets fault, 0=reset req'd to clear fault
   Cfg_OvrdPermIntlk : BOOL;   // 1=Override ignores Bypassable Perm/ Intlk; 0=always use Perm/Intlk
   Cfg_ShedOnFailToStart : BOOL := 1;   // 1=Stop Motor and Alarm on Fail to Start; 0=Alarm only on Fail to Start
   Cfg_ShedOnIOFault : BOOL := 1;   // 1=Stop Motor and Alarm on I/O Fault; 0=Alarm only on I/O Fault
   Cfg_SimScaleEU : BOOL;   // 1=In simulation, scale Speed Ref EU to Speed Fdbk EU
   Cfg_SimScaleRaw : BOOL;   // 1=In simulation, scale Speed Ref EU to raw, then raw to Speed Fdbk EU
   Cfg_HasFailToStartAlm : ALIAS FOR FailToStart.Cfg_Exists;   // 1=Fail to Start Alarm exists and will be checked
   Cfg_HasFailToStopAlm : ALIAS FOR FailToStop.Cfg_Exists;   // 1=Fail to Stop Alarm exists and will be checked
   Cfg_HasIntlkTripAlm : ALIAS FOR IntlkTrip.Cfg_Exists;   // 1=Interlock Trip Alarm exists and will be checked
   Cfg_HasDriveFaultAlm : ALIAS FOR DriveFault.Cfg_Exists;   // 1=Drive Fault alarm exists and will be checked
   Cfg_HasIOFaultAlm : ALIAS FOR IOFault.Cfg_Exists;   // 1=I/O Fault Alarm exists and will be checked
   Cfg_FailToStartResetReqd : ALIAS FOR FailToStart.Cfg_ResetReqd;   // 1=Reset requied to clear Fail to Start Alarm
   Cfg_FailToStopResetReqd : ALIAS FOR FailToStop.Cfg_ResetReqd;   // 1=Reset required to clear Fail to Stop Alarm
   Cfg_IntlkTripResetReqd : ALIAS FOR IntlkTrip.Cfg_ResetReqd;   // 1=Reset required to clear Interlock Trip Alarm
   Cfg_DriveFaultResetReqd : ALIAS FOR DriveFault.Cfg_ResetReqd;   // 1=Reset required to clear Drive Fault Alarm
   Cfg_IOFaultResetReqd : ALIAS FOR IOFault.Cfg_ResetReqd;   // 1=Reset required to clear I/O Fault Alarm
   Cfg_FailToStartAckReqd : ALIAS FOR FailToStart.Cfg_AckReqd;   // 1=Acknowledge required for Fail to Start Alarm
   Cfg_FailToStopAckReqd : ALIAS FOR FailToStop.Cfg_AckReqd;   // 1=Acknowledge required for Fail to Stop Alarm
   Cfg_IntlkTripAckReqd : ALIAS FOR IntlkTrip.Cfg_AckReqd;   // 1=Acknowledge required for Interlock Trip Alarm
   Cfg_DriveFaultAckReqd : ALIAS FOR DriveFault.Cfg_AckReqd;   // 1=Acknowledge required for Drive Fault Alarm
   Cfg_IOFaultAckReqd : ALIAS FOR IOFault.Cfg_AckReqd;   // 1=Acknowledge required for I/O Fault Alarm
   Cfg_FailToStartSeverity : ALIAS FOR FailToStart.Cfg_Severity;   // Fail To Start Alarm Severity: 1..250=Low, 251..500=Medium, 501..750=High, 751..1000=Urgent
   Cfg_FailToStopSeverity : ALIAS FOR FailToStop.Cfg_Severity;   // Fail To Stop Alarm Severity: 1..250=Low, 251..500=Medium, 501..750=High, 751..1000=Urgent
   Cfg_IntlkTripSeverity : ALIAS FOR IntlkTrip.Cfg_Severity;   // Interlock Trip Alarm Severity: 1..250=Low, 251..500=Medium, 501..750=High, 751..1000=Urgent
   Cfg_DriveFaultSeverity : ALIAS FOR DriveFault.Cfg_Severity;   // Drive Fault Alarm Severity: 1..250=Low, 251..500=Medium, 501..750=High, 751..1000=Urgent
   Cfg_IOFaultSeverity : ALIAS FOR IOFault.Cfg_Severity;   // I/O Fault Alarm Severity: 1..250=Low, 251..500=Medium, 501..750=High, 751..1000=Urgent
   Cfg_MinSpdRef : REAL;   // Minimum Speed Reference in EU (for limiting)
   Cfg_MaxSpdRef : REAL := 60.0;   // Maximum Speed Reference in EU (for limiting)
   Cfg_SpeedRefRawMin : INT;   // Speed Reference Minimum in Drive (raw) Units (for scaling)
   Cfg_SpeedRefRawMax : INT := 6000;   // Speed Reference Maximum in Drive (raw) Units (for scaling)
   Cfg_SpeedRefEUMin : REAL;   // Speed Reference Minimum in Engineering Units (for scaling)
   Cfg_SpeedRefEUMax : REAL := 60.0;   // Speed Reference Maximum in Engineering Units (for scaling)
   Cfg_SpeedFdbkRawMin : INT;   // Speed Feedback Minimum in Drive (raw) Units (for scaling)
   Cfg_SpeedFdbkRawMax : INT := 6000;   // Speed Feedback Maximum in Drive (raw) Units (for scaling)
   Cfg_SpeedFdbkEUMin : REAL;   // Speed Feedback Minimum in Engineering Units (for scaling)
   Cfg_SpeedFdbkEUMax : REAL := 60.0;   // Speed Feedback Maximum in Engineering Units (for scaling)
   Cfg_SimRampT : DINT := 10;   // Time to ramp speed fdbk when in Simulation (sec)
   Cfg_FailToStartT : DINT := 15;   // Time after Start to get Run Feedback before Fault (sec)
   Cfg_FailToStopT : DINT := 15;   // Time after Stop to drop Run Feedback before Fault (sec)
   Cfg_ResetPulseT : DINT := 2;   // Time to pulse Out_Reset to clear drive fault
   Cfg_MaxJogT : REAL;   // Maximum jog time (sec, 0=unlimited)
   Cfg_OperKeep : SINT;   // Oper keeps control in Prog Mode: .0=Reference, .1=Start/Stop, .2=Fwd/Rev
   Cfg_ProgKeep : SINT;   // Prog keeps control in Oper Mode: .0=Reference, .1=Start/Stop, .2=Fwd/Rev
   PSet_SpeedRef : REAL;   // Program Setting of Speed Reference (EU)
   PSet_Owner : DINT;   // Program Owner Request ID (non-zero) or Release (zero)
   OSet_SpeedRef : REAL;   // Operator Setting of Speed Reference (EU)
   PCmd_Start : BOOL;   // Program Command to Start Drive
   PCmd_Stop : BOOL;   // Program Command to Stop Drive
   PCmd_Fwd : BOOL;   // Program Command to set direction to Fowrard
   PCmd_Rev : BOOL;   // Program Command to set direction to Reverse
   PCmd_Acq : ALIAS FOR Mode.PCmd_Acq;
   PCmd_Rel : ALIAS FOR Mode.PCmd_Rel;
   PCmd_Lock : ALIAS FOR Mode.PCmd_Lock;
   PCmd_Unlock : ALIAS FOR Mode.PCmd_Unlock;
   PCmd_Reset : BOOL;   // Program Command to Reset drive fault and all Alarms requiring Reset
   PCmd_FailToStartAck : ALIAS FOR FailToStart.PCmd_Ack;   // Program Command to Acknowledge Fail to Start Alarm
   PCmd_FailToStartSuppress : ALIAS FOR FailToStart.PCmd_Suppress;   // Program Command to Suppress Fail to Start Alarm
   PCmd_FailToStartUnsuppress : ALIAS FOR FailToStart.PCmd_Unsuppress;   // Program Command to Unsuppress Fail to Start Alarm
   PCmd_FailToStartUnshelve : ALIAS FOR FailToStart.PCmd_Unshelve;   // Program Command to Unshelve Fail to Start Alarm
   PCmd_FailToStopAck : ALIAS FOR FailToStop.PCmd_Ack;   // Program Command to Acknowledge Fail to Stop Alarm
   PCmd_FailToStopSuppress : ALIAS FOR FailToStop.PCmd_Suppress;   // Program Command to Suppress Fail to Stop Alarm
   PCmd_FailToStopUnsuppress : ALIAS FOR FailToStop.PCmd_Unsuppress;   // Program Command to Unsuppress Fail to Stop Alarm
   PCmd_FailToStopUnshelve : ALIAS FOR FailToStop.PCmd_Unshelve;   // Program Command to Unshelve Fail to Stop Alarm
   PCmd_IntlkTripAck : ALIAS FOR IntlkTrip.PCmd_Ack;   // Program Command to Acknowledge Interlock Trip Alarm
   PCmd_IntlkTripSuppress : ALIAS FOR IntlkTrip.PCmd_Suppress;   // Program Command to Suppress Interlock Trip Alarm
   PCmd_IntlkTripUnsuppress : ALIAS FOR IntlkTrip.PCmd_Unsuppress;   // Program Command to Unsuppress Interlock Trip Alarm
   PCmd_IntlkTripUnshelve : ALIAS FOR IntlkTrip.PCmd_Unshelve;   // Program Command to Unshelve Interlock Trip Alarm
   PCmd_DriveFaultAck : ALIAS FOR DriveFault.PCmd_Ack;   // Program Command to Acknowledge Drive Fault Alarm
   PCmd_DriveFaultSuppress : ALIAS FOR DriveFault.PCmd_Suppress;   // Program Command to Suppress Drive Fault Alarm
   PCmd_DriveFaultUnsuppress : ALIAS FOR DriveFault.PCmd_Unsuppress;   // Program Command to Unsuppress Drive Fault Alarm
   PCmd_DriveFaultUnshelve : ALIAS FOR DriveFault.PCmd_Unshelve;   // Program Command to Unshelve Drive Fault Alarm
   PCmd_IOFaultAck : ALIAS FOR IOFault.PCmd_Ack;   // Program Command to Acknowledge I/O Fault Alarm
   PCmd_IOFaultSuppress : ALIAS FOR IOFault.PCmd_Suppress;   // Program Command to Suppress I/O Fault Alarm
   PCmd_IOFaultUnsuppress : ALIAS FOR IOFault.PCmd_Unsuppress;   // Program Command to Unsuppress I/O Fault Alarm
   PCmd_IOFaultUnshelve : ALIAS FOR IOFault.PCmd_Unshelve;   // Program Command to Unshelve I/O Fault Alarm
   OCmd_Start : BOOL;   // Operator Command to Start Drive
   OCmd_Stop : BOOL;   // Operator Command to Stop Drive
   OCmd_Jog : BOOL;   // Operator Command to Jog Drive (not cleared by P_PF52x!)
   OCmd_Fwd : BOOL;   // Operator Command to set direction to Forward
   OCmd_Rev : BOOL;   // Operator Command to set direction to Reverse
   OCmd_Bypass : BOOL;   // Operator Command to Bypass all Bypassable Interlocks and Permissives
   OCmd_Check : BOOL;   // Operator Command to Check (not bypass) all Interlocks and Permissives
   MCmd_Disable : BOOL;   // Maintenance Command to Disable Drive
   MCmd_Enable : BOOL;   // Maintenance Command to Enable (allow to run) Drive
   MCmd_Acq : ALIAS FOR Mode.MCmd_Acq;
   MCmd_Rel : ALIAS FOR Mode.MCmd_Rel;
   OCmd_AcqLock : ALIAS FOR Mode.OCmd_AcqLock;
   OCmd_Unlock : ALIAS FOR Mode.OCmd_UnlockRel;
   OCmd_Reset : BOOL;   // Operator Command to Reset all Alarms requiring Reset
   OCmd_ResetAckAll : BOOL;   // Operator Command to Reset all Alarms and latched Shed conditions
END_VAR
VAR_OUTPUT
   Val_SpeedRef : REAL; {access Read Only, visible}   // Speed Reference (target) to drive
   Val_SpeedFdbk : REAL; {access Read Only, visible}   // Speed Feedback (actual) from drive
   Val_SpeedRefRaw : REAL; {access Read Only}   // Copy of Speed Reference Output (in Raw units) for faceplate
   Val_SpeedFdbkRaw : REAL; {access Read Only}   // Copy of Speed Feedback Input (in Raw units) for faceplate
   Val_SpeedRefEUMin : REAL; {access Read Only}   // Minimum of Speed Reference = MIN (Cfg_SpeedFdbkEUMin, Cfg_SpeedFdbkEUMax)
   Val_SpeedRefEUMax : REAL := 130.0; {access Read Only}   // Maximum of Speed Reference = MAX (Cfg_SpeedFdbkEUMin, Cfg_SpeedFdbkEUMax)
   Val_SpeedFdbkEUMin : REAL; {access Read Only}   // Minimum of Speed Feedback = MIN (Cfg_SpeedFdbkEUMin, Cfg_SpeedFdbkEUMax)
   Val_SpeedFdbkEUMax : REAL := 130.0; {access Read Only}   // Maximum of Speed Feedback = MAX (Cfg_SpeedFdbkEUMin, Cfg_SpeedFdbkEUMax)
   Val_LastFaultCode : DINT; {access Read Only}   // Last drive fault code (enum) (Par 951)
   Val_OutCurrent : REAL; {access Read Only}   // Drive output current (Amps)
   Val_OutPower : REAL; {access Read Only}   // Drive output power (kW)
   SrcQ_IO : SINT; {access Read Only}   // Source and Quality of primary I/O (enumeration)
   SrcQ : SINT; {access Read Only}   // Source and Quality of primary Val/Sts (enumeration)
   Val_Cmd : SINT; {access Read Only}   // Device Command 0=None, 1=Stop, 2=StartFwd 3=StartRev 4=JogFwd 5=JogRev
   Val_Fdbk : SINT; {access Read Only}   // Device Feedback 0=Stopped, 1=Running Fwd 2=Running Rev 3=Accelerating 4=Decelerating
   Val_Sts : SINT; {access Read Only}   // Device Confirmed Sts 0? 1=Stop 2=RunF 3=RunR 4=JogF 5=JogR 6=Stopping 7=Starting F 8=Starting R, 33=Disabled
   Val_Fault : SINT; {access Read Only, visible}   // Device Fault Status 0=None, 16=Fail to Start, 17 = Fail to Stop, 18=Drive Fault, 32=I/O Fault, 34=Config Error
   Val_Mode : ALIAS FOR Mode.Val; {access Read Only}
   Val_Owner : DINT; {access Read Only}   // Current Object Owner ID (0=not owned)
   Val_Notify : SINT; {access Read Only}   // Current Alarm Level and Acknowledgement (enumeration)
   Sts_Stopped : BOOL := 1; {access Read Only, visible}   // 1=Drive requested to stop and is confirmed stopped
   Sts_Starting : BOOL; {access Read Only, visible}   // 1=Drive requested to run and awaiting run feedback
   Sts_Running : BOOL; {access Read Only, visible}   // 1=Drive requested to run and is confirmed running
   Sts_Stopping : BOOL; {access Read Only, visible}   // 1=Drive requested to stop and awaiting stopped feedback
   Sts_Jogging : BOOL; {access Read Only, visible}   // 1=Drive requested to Jog
   Sts_CommandDir : BOOL := 1; {access Read Only}   // 1=Drive commanded to Forward, 0=Reverse
   Sts_ActualDir : BOOL := 1; {access Read Only, visible}   // 1=Drive Actual direction is Forward, 0=Reverse
   Sts_Accel : BOOL; {access Read Only}   // 1=Drive is Accelerating
   Sts_Decel : BOOL; {access Read Only}   // 1=Drive is Decelerating
   Sts_NotReady : BOOL; {access Read Only}   // 1=Device Not Ready, see detail bits for reason
   Sts_AtSpeed : BOOL; {access Read Only, visible}   // 1=Drive is running at reference speed
   Sts_SpeedLimited : BOOL; {access Read Only, visible}   // 1=Speed Reference Setting exceeds configured Max/Min limit
   Sts_DigIn1 : BOOL; {access Read Only}   // Drive Digital Input 1 Status
   Sts_DigIn2 : BOOL; {access Read Only}   // Drive Digital Input 2 Status
   Sts_DigIn3 : BOOL; {access Read Only}   // Drive Digital Input 3 Status
   Sts_DigIn4 : BOOL; {access Read Only}   // Drive Digital Input 4 Status
   Sts_Available : BOOL; {access Read Only, visible}   // 1=Drive available for control by automation (Prog)
   Sts_Bypass : BOOL; {access Read Only}   // 1=Bypassable Interlocks and Permissives are Bypassed
   Sts_BypActive : BOOL; {access Read Only}   // 1=Bypassing Active (Bypassed or Maintenance)
   Sts_Disabled : BOOL; {access Read Only}   // 1=Drive is Disabled
   Sts_NotRdy : BOOL; {access Read Only}   // 1=Motor is Not Ready to Run (independent of Mode)
   Nrdy_Disabled : BOOL; {access Read Only}   // 1=Device Not Ready: Device Disabled by Maintenance
   Nrdy_CfgErr : BOOL; {access Read Only}   // 1=Device Not Ready: Configuration Error
   Nrdy_Intlk : BOOL; {access Read Only}   // 1=Device Not Ready: Interlock Not OK
   Nrdy_Perm : BOOL; {access Read Only}   // 1=Device Not Ready: Permissive Not OK
   Nrdy_OperPrio : BOOL; {access Read Only}   // 1=Device Not Ready: Operator State 0 Priority Command Requires Reset
   Nrdy_Fail : BOOL; {access Read Only}   // 1=Device Not Ready: Device Failure (Shed Requires Reset)
   Nrdy_IOFault : BOOL; {access Read Only}   // 1=Device Not Ready: I/O Fault (Shed Requires Reset)
   Nrdy_Trip : BOOL; {access Read Only}   // 1=Device not Ready: Deivce Tripped (Drive Fault)
   Nrdy_DriveNR : BOOL; {access Read Only}   // 1=Device Note Ready: Drive Not Ready
   Nrdy_NoMode : BOOL; {access Read Only}   // 1=Device Not Ready: Device Logic Disabled / NO Mode
   Sts_MaintByp : BOOL; {access Read Only}   // 1=A Maintenance Bypass is Active, display icon
   Sts_AlmInh : BOOL; {access Read Only}   // 1=An Alarm is Shelved, Disabled or Suppressed, display icon
   Sts_Err : BOOL; {access Read Only, visible}   // 1=Error in Config: see detail bits for reason
   Err_Timer : BOOL; {access Read Only}   // 1=Error in Config: Invalid Check or Reset Pulse Time (use 0 to 2147483)
   Err_Sim : BOOL; {access Read Only}   // 1=Error in Config: simulation timer preset: use 0 to 2147483)
   Err_Alarm : BOOL; {access Read Only}   // 1=Error in Config: Alarm Min On Time, Shelf Time, Severity
   Err_FdbkRaw : BOOL; {access Read Only}   // 1=Erron in Config: Speed Fdbk Raw Min = Max
   Err_FdbkEU : BOOL; {access Read Only}   // 1=Error in Config: Speed Fdbk EU Min = Max
   Err_RefLim : BOOL; {access Read Only}   // 1=Error in Config: Speed Ref Limit Min > Max
   Err_RefEU : BOOL; {access Read Only}   // 1=Error in Config: Speed Ref EU Min = Max
   Err_RefRaw : BOOL; {access Read Only}   // 1=Error in Config: Speed Ref Raw Min = Max
   Sts_Hand : ALIAS FOR Mode.Sts_Hand; {access Read Only, visible}
   Sts_Maint : ALIAS FOR Mode.Sts_Maint; {access Read Only, visible}
   Sts_Ovrd : ALIAS FOR Mode.Sts_Ovrd; {access Read Only, visible}
   Sts_Prog : ALIAS FOR Mode.Sts_Prog; {access Read Only, visible}
   Sts_Oper : ALIAS FOR Mode.Sts_Oper; {access Read Only, visible}
   Sts_ProgOperLock : ALIAS FOR Mode.Sts_ProgOperLock; {access Read Only}
   Sts_NoMode : ALIAS FOR Mode.Sts_NoMode; {access Read Only}
   Sts_MAcqRcvd : ALIAS FOR Mode.Sts_MAcqRcvd; {access Read Only}
   Sts_FailToStart : ALIAS FOR FailToStart.Inp;   // 1=Drive Failed to Start (One-Shot)
   Alm_FailToStart : ALIAS FOR FailToStart.Alm;   // 1=Drive Fail to Start Alarm
   Ack_FailToStart : ALIAS FOR FailToStart.Ack;   // 1=Fail to Start Alarm has been acknowledged
   Sts_FailToStartDisabled : ALIAS FOR FailToStart.Disabled;   // 1=Fail to Start Alarm has been Disabled by Maintenance
   Sts_FailToStartShelved : ALIAS FOR FailToStart.Shelved;   // 1=Fail to Start Alarm has been Shelved by Operator
   Sts_FailToStartSuppressed : ALIAS FOR FailToStart.Suppressed;   // 1=Fail to Start Alarm has been Suppressed by Program
   Sts_FailToStop : ALIAS FOR FailToStop.Inp;   // 1=Drive Failed to Stop
   Alm_FailToStop : ALIAS FOR FailToStop.Alm;   // 1=Drive Fail to Stop Alarm
   Ack_FailToStop : ALIAS FOR FailToStop.Ack;   // 1=Fail to Stop Alarm has been acknowledged
   Sts_FailToStopDisabled : ALIAS FOR FailToStop.Disabled;   // 1=Fail to Stop Alarm has been Disabled by Maintenance
   Sts_FailToStopShelved : ALIAS FOR FailToStop.Shelved;   // 1=Fail to Stop Alarm has been Shelved by Operator
   Sts_FailToStopSuppressed : ALIAS FOR FailToStop.Suppressed;   // 1=Fail to Stop Alarm has been Suppressed by Program
   Sts_IntlkTrip : ALIAS FOR IntlkTrip.Inp;   // 1=Drive was stopped by an Interlock NOT OK (One-Shot)
   Alm_IntlkTrip : ALIAS FOR IntlkTrip.Alm;   // 1=Alarm: Drive stopped by an Interlock NOT OK
   Ack_IntlkTrip : ALIAS FOR IntlkTrip.Ack;   // 1=Interlock Trip Alarm has been acknowledged
   Sts_IntlkTripDisabled : ALIAS FOR IntlkTrip.Disabled;   // 1=Interlock Trip Alarm has been Disabled by Maintenance
   Sts_IntlkTripShelved : ALIAS FOR IntlkTrip.Shelved;   // 1=Interlock Trip Alarm has been Shelved by Operator
   Sts_IntlkTripSuppressed : ALIAS FOR IntlkTrip.Suppressed;   // 1=Interlock Trip Alarm has been Suppressed by Program
   Sts_DriveFault : ALIAS FOR DriveFault.Inp;   // 1=Drive Fault (see drive display or manual)
   Alm_DriveFault : ALIAS FOR DriveFault.Alm;   // 1=Alarm: Drive Fault (see drive display or manual)
   Ack_DriveFault : ALIAS FOR DriveFault.Ack;   // 1=Drive Fault Alarm has been acknowledged
   Sts_DriveFaultDisabled : ALIAS FOR DriveFault.Disabled;   // 1=Drive Fault Alarm has been Disabled by Maintenance
   Sts_DriveFaultShelved : ALIAS FOR DriveFault.Shelved;   // 1=Drive Fault Alarm has been Shelved by Operator
   Sts_DriveFaultSuppressed : ALIAS FOR DriveFault.Suppressed;   // 1=Drive Fault Alarm has been Suppressed by Program
   Sts_IOFault : ALIAS FOR IOFault.Inp;   // I/O Comm Fault Status (0=OK, 1=Bad)
   Alm_IOFault : ALIAS FOR IOFault.Alm;   // 1=I/O Fault Alarm
   Ack_IOFault : ALIAS FOR IOFault.Ack;   // 1=I/O Fault Alarm has been acknowledged
   Sts_IOFaultDisabled : ALIAS FOR IOFault.Disabled;   // 1=I/O Fault Alarm has been Disabled by Maintenance
   Sts_IOFaultShelved : ALIAS FOR IOFault.Shelved;   // 1=I/O Fault Alarm has been Shelved by Operator
   Sts_IOFaultSuppressed : ALIAS FOR IOFault.Suppressed;   // 1=I/O Fault Alarm has been Suppressed by Program
   Rdy_Start : BOOL; {access Read Only}   // 1=Ready to receive OCmd_Start (enables HMI button)
   Rdy_Stop : BOOL; {access Read Only}   // 1=Ready to receive OCmd_Stop (enables HMI button)
   Rdy_Jog : BOOL; {access Read Only}   // 1=Ready to receive OCmd_Jog (enables HMI button)
   Rdy_Fwd : BOOL; {access Read Only}   // 1=Ready to receive OCmd_Fwd (enabled HMI button)
   Rdy_Rev : BOOL; {access Read Only}   // 1=Ready to receive OCmd_Rev (enables HMI button)
   Rdy_Bypass : BOOL; {access Read Only}   // 1=Ready to receive OCmd_Bypass (enables HMI button)
   Rdy_Check : BOOL; {access Read Only}   // 1=Ready to receive OCmd_Check (enables HMI button)
   Rdy_Disable : BOOL; {access Read Only}   // 1=Ready to receive MCmd_Disable (enables HMI button)
   Rdy_Enable : BOOL; {access Read Only}   // 1=Ready to receive MCmd_Enable (enables HMI button)
   Rdy_Reset : BOOL; {access Read Only}   // 1=Ready to receive OCmd_Reset (enables HMI button)
   Rdy_ResetAckAll : BOOL; {access Read Only}   // 1=At least one Alarm or latched Shed condition requires Reset or Ack
   Rdy_SpeedRef : BOOL; {access Read Only}   // 1=Ready to receive OSet_SpeedRef (enables data entry field)
   P_PF52x : BOOL;   // Unique Parameter Name for auto - discovery
END_VAR
VAR
   Mode : P_Mode := (Cfg_PCmdClear := 1, Cfg_OvrdOverLock := 1, Rdy_OAcq := 1);   // Drive Mode Selection
   IOFault : P_Alarm := (Cfg_AckReqd := 1, Cfg_AllowShelve := 1, Cfg_AllowDisable := 1, Cfg_PCmdClear := 1, Cfg_Severity := 1000, Cfg_AlmMinOnT := 5, PCfg_AllowExist := 1, Ack := 1);   // I/O Fault Alarm
   IntlkTrip : P_Alarm := (Cfg_AckReqd := 1, Cfg_AllowShelve := 1, Cfg_AllowDisable := 1, Cfg_PCmdClear := 1, Cfg_Severity := 500, Cfg_AlmMinOnT := 5, PCfg_AllowExist := 1, Ack := 1);   // Interlock Trip Alarm
   FailToStop : P_Alarm := (Cfg_AckReqd := 1, Cfg_AllowShelve := 1, Cfg_AllowDisable := 1, Cfg_PCmdClear := 1, Cfg_Severity := 1000, Cfg_AlmMinOnT := 5, PCfg_AllowExist := 1, Ack := 1);   // Drive Failed to Stop Alarm
   FailToStart : P_Alarm := (Cfg_AckReqd := 1, Cfg_AllowShelve := 1, Cfg_AllowDisable := 1, Cfg_PCmdClear := 1, Cfg_Severity := 1000, Cfg_AlmMinOnT := 5, PCfg_AllowExist := 1, Ack := 1);   // Drive Failed to Start Alarm
   Cfg_Tag : STRING_20 := 'P_PF52x';   // Tagname for display on HMI
   Cfg_Label : STRING_20 := 'Motor Speed Control';   // Label for graphic symbol displayed on HMI
   Cfg_Desc : STRING_40 := 'PF523 / PF525 Variable Frequency Drive';   // Description for display on HMI
   Wrk_Run : BOOL; {access None}   // 1=Drive should be "running", 0=should be "stopped"
   Wrk_StartRetrigT : TIMER; {access None}   // Time to pulse start output on start command retrigger (Maint)
   Wrk_StopRetrigT : TIMER; {access None}   // Time to pulse stop output on stop command retrigger (Maint)
   Wrk_RunFdbk : BOOL; {access None}   // Run Feedback based on mode, simulation, etc. 1=running
   Wrk_Notify : DINT; {access None}   // Buffer for building Val_Notify
   Wrk_Bypass : BOOL; {access None}   // Internal Bypassable Permissives and Interlocks are Bypassed flag
   Wrk_Disabled : BOOL; {access None}   // Internal Drive is Disabled
   DriveFault : P_Alarm := (Cfg_AckReqd := 1, Cfg_AllowShelve := 1, Cfg_AllowDisable := 1, Cfg_PCmdClear := 1, Cfg_Severity := 1000, Cfg_AlmMinOnT := 5, PCfg_AllowExist := 1, Ack := 1);   // Drive Faulted Alarm
   Cfg_SpeedRefEU : STRING_8 := 'Hz';   // Speed Reference Engineering Units for display on HMI
   Wrk_SpeedRef : REAL; {access None}   // Working copy of Speed Reference (for limiting)
   Wrk_Rev : BOOL; {access None}   // Working (internal) Direction 1=Reverse 0=Forward (default)
   Wrk_Jog : BOOL; {access None}   // 1=Jog Drive, 0=Drive not jogging
   Wrk_ResetT : TIMER; {access None}   // Reset Output Pulse Timer
   Wrk_ResetONS : BOOL; {access None}   // One-Shot to fire Reset Timer to ensure min. output ON time.
   Cfg_SpeedFdbkEU : STRING_8 := 'Hz';   // Speed Feedback Engineering Units for display on HMI
   Cfg_RevText : STRING_16 := 'Reverse';   // Name for Reverse Direction, e.g., "Down", "Reverse"
   Cfg_FwdText : STRING_16 := 'Forward';   // Name for Forward Direction, e.g., "Up", "Forward"
   Wrk_StopT : TIMER; {access None}   // Stop Check Timer (for Fail to Stop)
   Wrk_StartT : TIMER; {access None}   // Start Check Timer (for Fail to Start)
   Inf_Tab : SINT;   // Tab to display (FTView ME)
   Wrk_Cmd : SINT; {access None}   // Buffer for building Val_Cmd
   Wrk_Sts : SINT; {access None}   // Buffer for building Val_Sts
   Wrk_Fault : SINT; {access None}   // Buffer for building Val_Fault
   Wrk_Retrigger : BOOL; {access None}   // Maint Start issued while running or Stop while stopped
   Wrk_Step : REAL; {access None}   // Amount to change simulated Speed Fdbk this scan (ramp)
   Wrk_ScanTime : REAL; {access None}   // Seconds since previous scan
   Wrk_ScanT : TIMER := (PRE := 2147483647); {access None}   // Scan Timer (milliseconds, always runs)
   Wrk_SimFdbkTgt : REAL; {access None}   // Speed Ref converted to Speed Fdbk units for simulation: target speed fdbk
   Inf_Type : STRING_16 := 'P_PF52x'; {access Read Only}   // Type identifier for HMI navigation
   Wrk_JogT : TIMER; {access None}   // Jog Timer
   Wrk_FaultDescFSC : CONTROL := (LEN := 1); {access None}   // FSC control for Fault Code List search
   Val_FaultDesc : STRING_40; {access Read Only}   // Description of Drive Fault (given LastFaultCode)
   Wrk_NotRdy : BOOL; {access None}   // Not Ready to run drive, assert Out_Stop
   Wrk_ProgKeep2ONS : BOOL; {access None}   // Prog Keep bit 2 one-shot store
   Wrk_ProgKeep1ONS : BOOL; {access None}   // Prog Keep bit 1 one-shot store
   Wrk_ProgKeep0ONS : BOOL; {access None}   // Prog Keep bit 0 one-shot store
   Wrk_OperKeep2ONS : BOOL; {access None}   // Oper Keep bit 2 one-shot store
   Wrk_OperKeep1ONS : BOOL; {access None}   // Oper Keep bit 1 one-shot store
   Wrk_OperKeep0ONS : BOOL; {access None}   // Oper Keep bit 0 one-shot store
   Inf_Lib : STRING_12 := 'RA-BAS'; {access Read Only}   // Display Library for Faceplate call-up
   Wrk_SrcQ : SINT; {access None}   // Register for building Source / Quality enumeration
   Cfg_DigIn4Txt : STRING_20 := 'Digital Input 4';   // Drive Digital Input 4 Label
   Cfg_DigIn3Txt : STRING_20 := 'Digital Input 3';   // Drive Digital Input 3 Label
   Cfg_DigIn2Txt : STRING_20 := 'Digital Input 2';   // Drive Digital Input 2 Label
   Cfg_DigIn1Txt : STRING_20 := 'Digital Input 1';   // Drive Digital Input 1 Label
   Wrk_NotRdyONS : BOOL; {access None}   // Assert Stop on One-Shot of Sts_NotRdy
END_VAR

ROUTINE EnableInFalse   (* ladder *)
// Disabled is asserted; Outputs OFF; Run Status shown but Alarms disabled
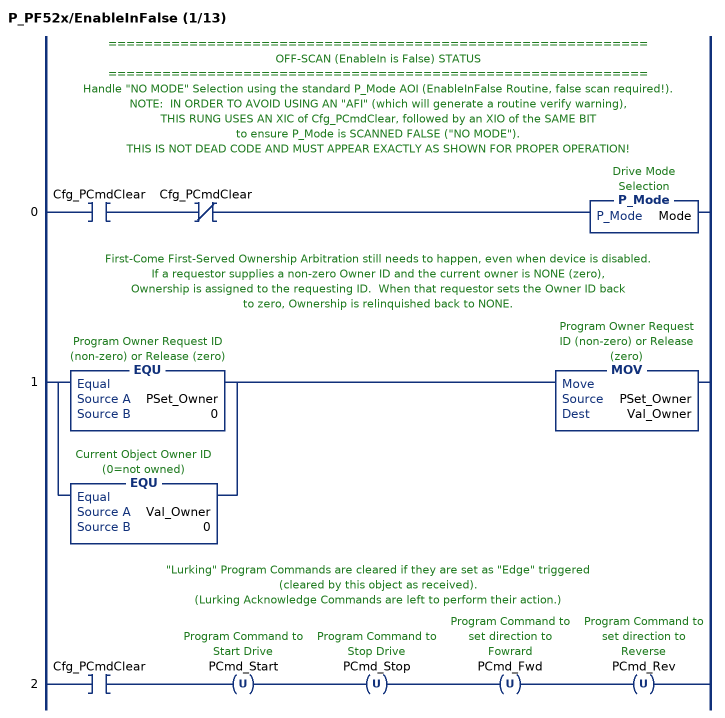
   // ============================================================
   // OFF-SCAN (EnableIn is False) STATUS
   // ============================================================
   // Handle "NO MODE" Selection using the standard P_Mode AOI (EnableInFalse Routine, false scan required!).
   // NOTE:  IN ORDER TO AVOID USING AN "AFI" (which will generate a routine verify warning),
   // THIS RUNG USES AN XIC of Cfg_PCmdClear, followed by an XIO of the SAME BIT
   // to ensure P_Mode is SCANNED FALSE ("NO MODE").
   // THIS IS NOT DEAD CODE AND MUST APPEAR EXACTLY AS SHOWN FOR PROPER OPERATION!
   0: XIC(Cfg_PCmdClear)XIO(Cfg_PCmdClear)P_Mode(Mode);
   // First-Come First-Served Ownership Arbitration still needs to happen, even when device is disabled.
   // If a requestor supplies a non-zero Owner ID and the current owner is NONE (zero),
   // Ownership is assigned to the requesting ID.  When that requestor sets the Owner ID back
   // to zero, Ownership is relinquished back to NONE.
   1: [EQU(PSet_Owner,0) ,EQU(Val_Owner,0) ]MOV(PSet_Owner,Val_Owner);
   // "Lurking" Program Commands are cleared if they are set as "Edge" triggered
   // (cleared by this object as received).
   // (Lurking Acknowledge Commands are left to perform their action.)
   2: XIC(Cfg_PCmdClear)OTU(PCmd_Start)OTU(PCmd_Stop)OTU(PCmd_Fwd)OTU(PCmd_Rev);
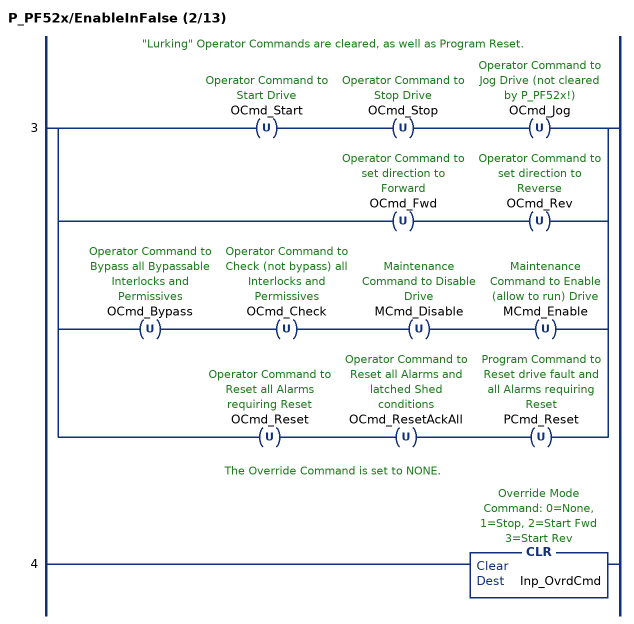
   // "Lurking" Operator Commands are cleared, as well as Program Reset.
   3: [OTU(OCmd_Start) OTU(OCmd_Stop) OTU(OCmd_Jog) ,OTU(OCmd_Fwd) OTU(OCmd_Rev) ,OTU(OCmd_Bypass) OTU(OCmd_Check) OTU(MCmd_Disable) OTU(MCmd_Enable) ,OTU(OCmd_Reset) OTU(OCmd_ResetAckAll) OTU(PCmd_Reset) ];
   // The Override Command is set to NONE.
   4: CLR(Inp_OvrdCmd);
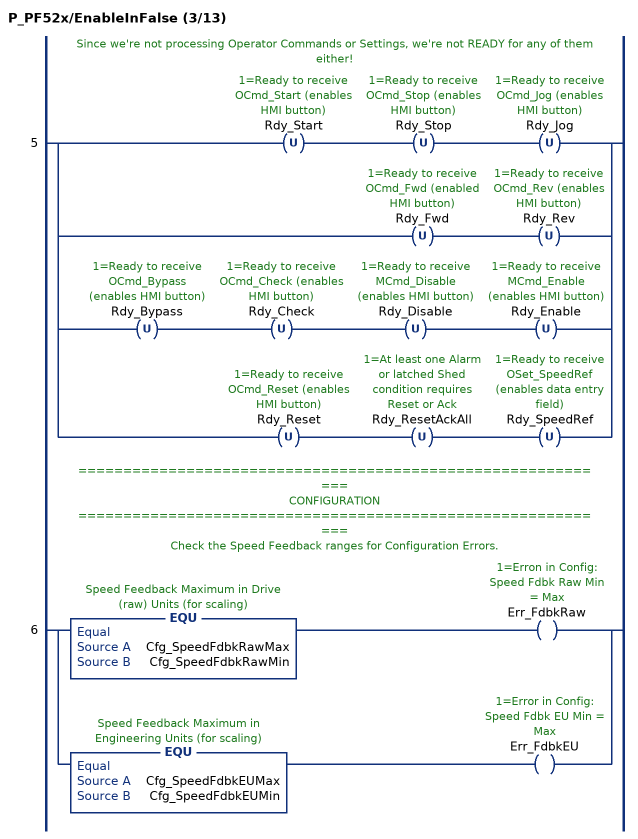
   // Since we're not processing Operator Commands or Settings, we're not READY for any of them either!
   5: [OTU(Rdy_Start) OTU(Rdy_Stop) OTU(Rdy_Jog) ,OTU(Rdy_Fwd) OTU(Rdy_Rev) ,OTU(Rdy_Bypass) OTU(Rdy_Check) OTU(Rdy_Disable) OTU(Rdy_Enable) ,OTU(Rdy_Reset) OTU(Rdy_ResetAckAll) OTU(Rdy_SpeedRef) ];
   // ============================================================
   // CONFIGURATION
   // ============================================================
   // Check the Speed Feedback ranges for Configuration Errors.
   6: [EQU(Cfg_SpeedFdbkRawMax,Cfg_SpeedFdbkRawMin) OTE(Err_FdbkRaw) ,EQU(Cfg_SpeedFdbkEUMax,Cfg_SpeedFdbkEUMin) OTE(Err_FdbkEU) ];
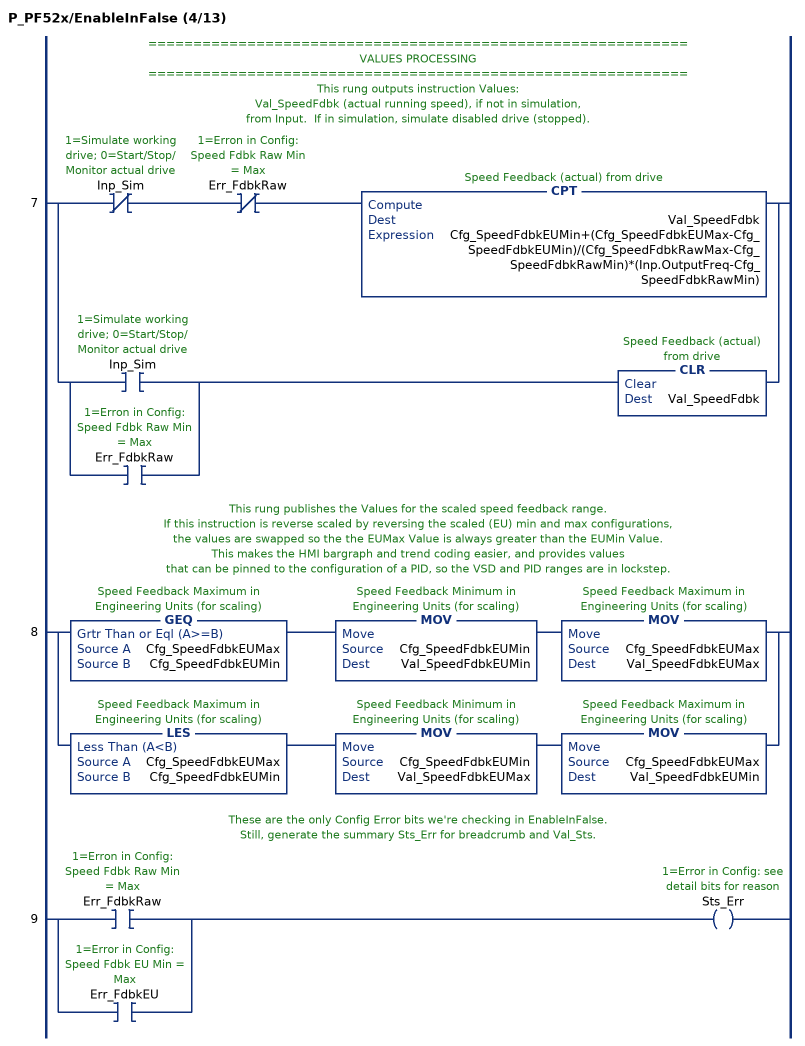
   // ============================================================
   // VALUES PROCESSING
   // ============================================================
   // This rung outputs instruction Values:
   // Val_SpeedFdbk (actual running speed), if not in simulation,
   // from Input.  If in simulation, simulate disabled drive (stopped).
   7: [XIO(Inp_Sim) XIO(Err_FdbkRaw) CPT(Val_SpeedFdbk,Cfg_SpeedFdbkEUMin+(Cfg_SpeedFdbkEUMax-Cfg_SpeedFdbkEUMin)/(Cfg_SpeedFdbkRawMax-Cfg_SpeedFdbkRawMin)*(Inp.OutputFreq-Cfg_SpeedFdbkRawMin)) ,[XIC(Inp_Sim) ,XIC(Err_FdbkRaw) ] CLR(Val_SpeedFdbk) ];
   // This rung publishes the Values for the scaled speed feedback range.
   // If this instruction is reverse scaled by reversing the scaled (EU) min and max configurations,
   // the values are swapped so the the EUMax Value is always greater than the EUMin Value.
   // This makes the HMI bargraph and trend coding easier, and provides values
   // that can be pinned to the configuration of a PID, so the VSD and PID ranges are in lockstep.
   8: [GEQ(Cfg_SpeedFdbkEUMax,Cfg_SpeedFdbkEUMin) MOV(Cfg_SpeedFdbkEUMin,Val_SpeedFdbkEUMin) MOV(Cfg_SpeedFdbkEUMax,Val_SpeedFdbkEUMax) ,LES(Cfg_SpeedFdbkEUMax,Cfg_SpeedFdbkEUMin) MOV(Cfg_SpeedFdbkEUMin,Val_SpeedFdbkEUMax) MOV(Cfg_SpeedFdbkEUMax,Val_SpeedFdbkEUMin) ];
   // These are the only Config Error bits we're checking in EnableInFalse.
   // Still, generate the summary Sts_Err for breadcrumb and Val_Sts.
   9: [XIC(Err_FdbkRaw) ,XIC(Err_FdbkEU) ]OTE(Sts_Err);
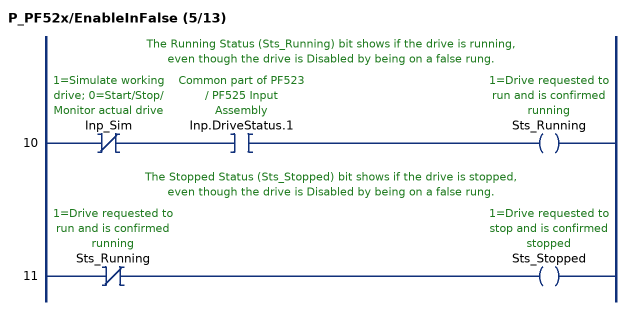
   // The Running Status (Sts_Running) bit shows if the drive is running,
   // even though the drive is Disabled by being on a false rung.
   10: XIO(Inp_Sim)XIC(Inp.DriveStatus.1)OTE(Sts_Running);
   // The Stopped Status (Sts_Stopped) bit shows if the drive is stopped,
   // even though the drive is Disabled by being on a false rung.
   11: XIO(Sts_Running)OTE(Sts_Stopped);
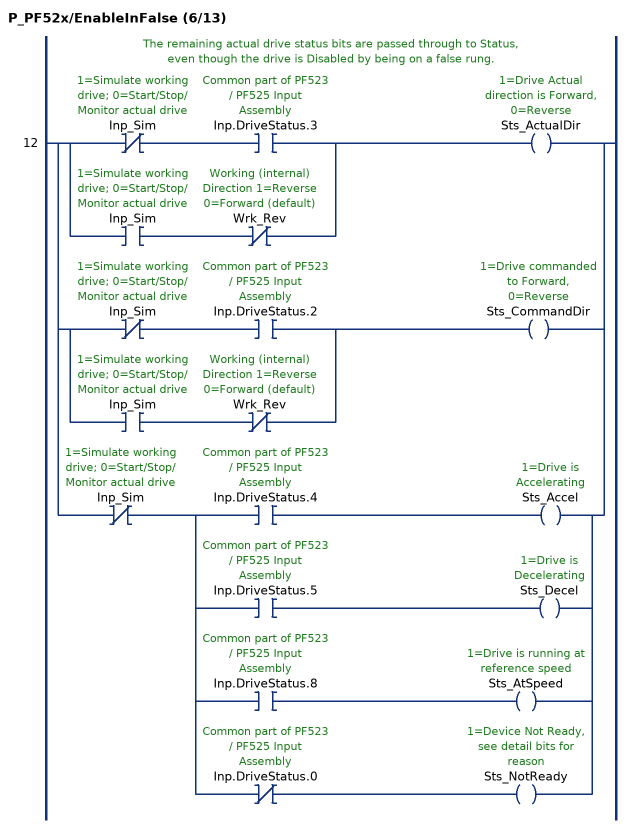
   // The remaining actual drive status bits are passed through to Status,
   // even though the drive is Disabled by being on a false rung.
   12: [[XIO(Inp_Sim) XIC(Inp.DriveStatus.3) ,XIC(Inp_Sim) XIO(Wrk_Rev) ] OTE(Sts_ActualDir) ,[XIO(Inp_Sim) XIC(Inp.DriveStatus.2) ,XIC(Inp_Sim) XIO(Wrk_Rev) ] OTE(Sts_CommandDir) ,XIO(Inp_Sim) [XIC(Inp.DriveStatus.4) OTE(Sts_Accel) ,XIC(Inp.DriveStatus.5) OTE(Sts_Decel) ,XIC(Inp.DriveStatus.8) OTE(Sts_AtSpeed) ,XIO(Inp.DriveStatus.0) OTE(Sts_NotReady) ] ];
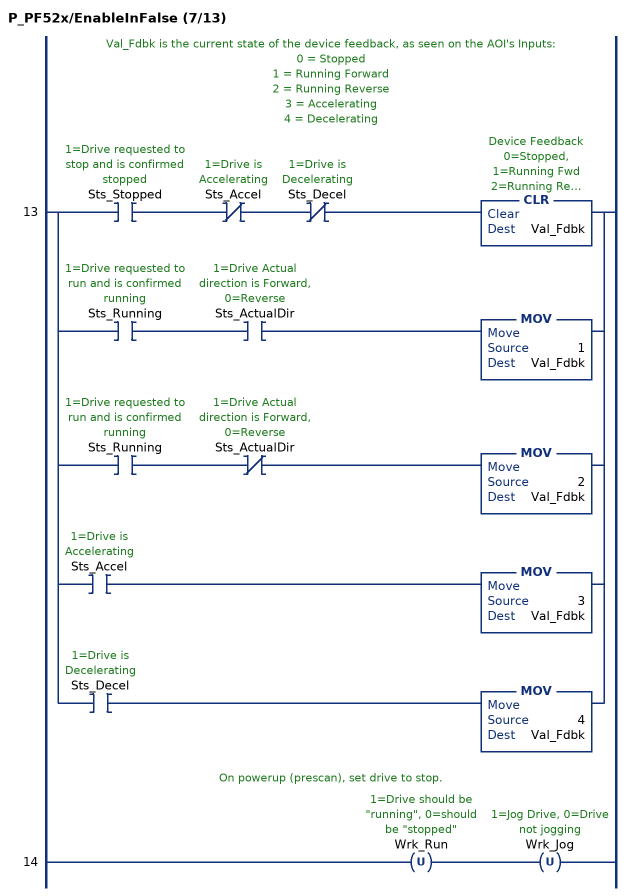
   // Val_Fdbk is the current state of the device feedback, as seen on the AOI's Inputs:
   // 0 = Stopped
   // 1 = Running Forward
   // 2 = Running Reverse
   // 3 = Accelerating
   // 4 = Decelerating
   13: [XIC(Sts_Stopped) XIO(Sts_Accel) XIO(Sts_Decel) CLR(Val_Fdbk) ,XIC(Sts_Running) XIC(Sts_ActualDir) MOV(1,Val_Fdbk) ,XIC(Sts_Running) XIO(Sts_ActualDir) MOV(2,Val_Fdbk) ,XIC(Sts_Accel) MOV(3,Val_Fdbk) ,XIC(Sts_Decel) MOV(4,Val_Fdbk) ];
   // On powerup (prescan), set drive to stop.
   14: OTU(Wrk_Run)OTU(Wrk_Jog);
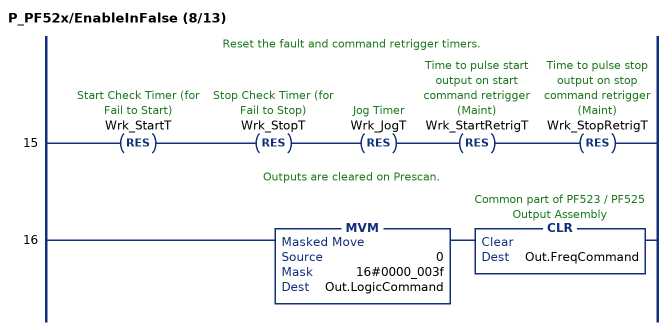
   // Reset the fault and command retrigger timers.
   15: RES(Wrk_StartT)RES(Wrk_StopT)RES(Wrk_JogT)RES(Wrk_StartRetrigT)RES(Wrk_StopRetrigT);
   // Outputs are cleared on Prescan.
   16: MVM(0,16#0000_003f,Out.LogicCommand)CLR(Out.FreqCommand);
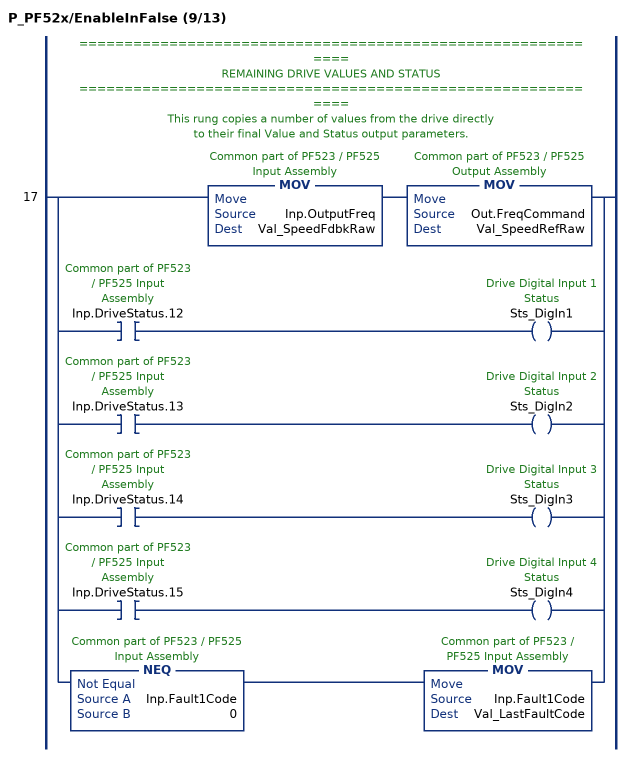
   // ============================================================
   // REMAINING DRIVE VALUES AND STATUS
   // ============================================================
   // This rung copies a number of values from the drive directly
   // to their final Value and Status output parameters.
   17: [MOV(Inp.OutputFreq,Val_SpeedFdbkRaw) MOV(Out.FreqCommand,Val_SpeedRefRaw) ,XIC(Inp.DriveStatus.12) OTE(Sts_DigIn1) ,XIC(Inp.DriveStatus.13) OTE(Sts_DigIn2) ,XIC(Inp.DriveStatus.14) OTE(Sts_DigIn3) ,XIC(Inp.DriveStatus.15) OTE(Sts_DigIn4) ,NEQ(Inp.Fault1Code,0) MOV(Inp.Fault1Code,Val_LastFaultCode) ];
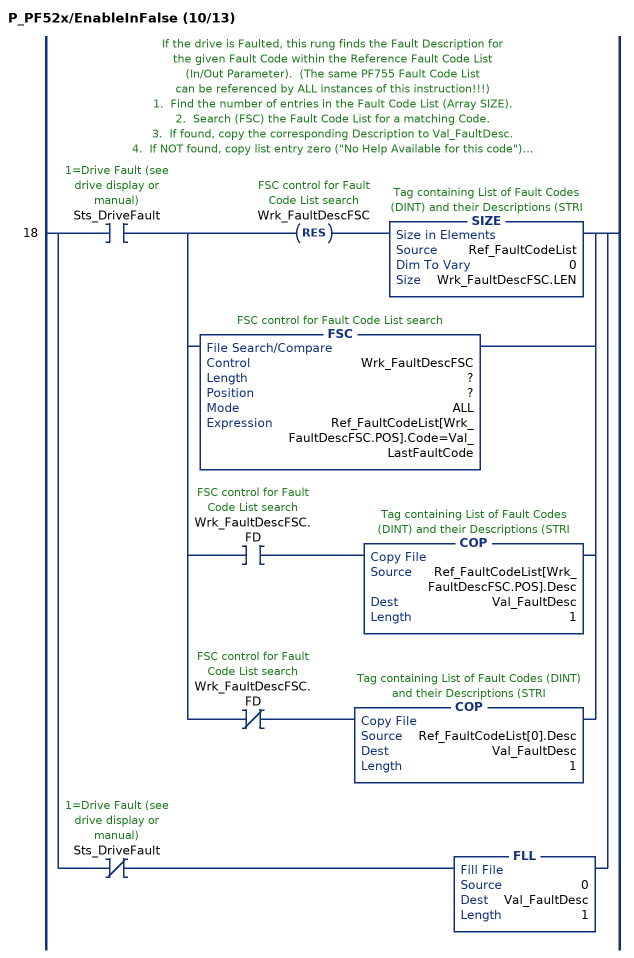
   // If the drive is Faulted, this rung finds the Fault Description for
   // the given Fault Code within the Reference Fault Code List
   // (In/Out Parameter).  (The same PF755 Fault Code List
   // can be referenced by ALL instances of this instruction!!!)
   // 1.  Find the number of entries in the Fault Code List (Array SIZE).
   // 2.  Search (FSC) the Fault Code List for a matching Code.
   // 3.  If found, copy the corresponding Description to Val_FaultDesc.
   // 4.  If NOT found, copy list entry zero ("No Help Available for this code").
   // And if the drive is not faulted, clear the Val_FaultDesc string.
   18: [XIC(Sts_DriveFault) [RES(Wrk_FaultDescFSC) SIZE(Ref_FaultCodeList,0,Wrk_FaultDescFSC.LEN) ,FSC(Wrk_FaultDescFSC,?,?,ALL,Ref_FaultCodeList[Wrk_FaultDescFSC.POS].Code=Val_LastFaultCode) ,XIC(Wrk_FaultDescFSC.FD) COP(Ref_FaultCodeList[Wrk_FaultDescFSC.POS].Desc,Val_FaultDesc,1) ,XIO(Wrk_FaultDescFSC.FD) COP(Ref_FaultCodeList[0].Desc,Val_FaultDesc,1) ] ,XIO(Sts_DriveFault) FLL(0,Val_FaultDesc,1) ];
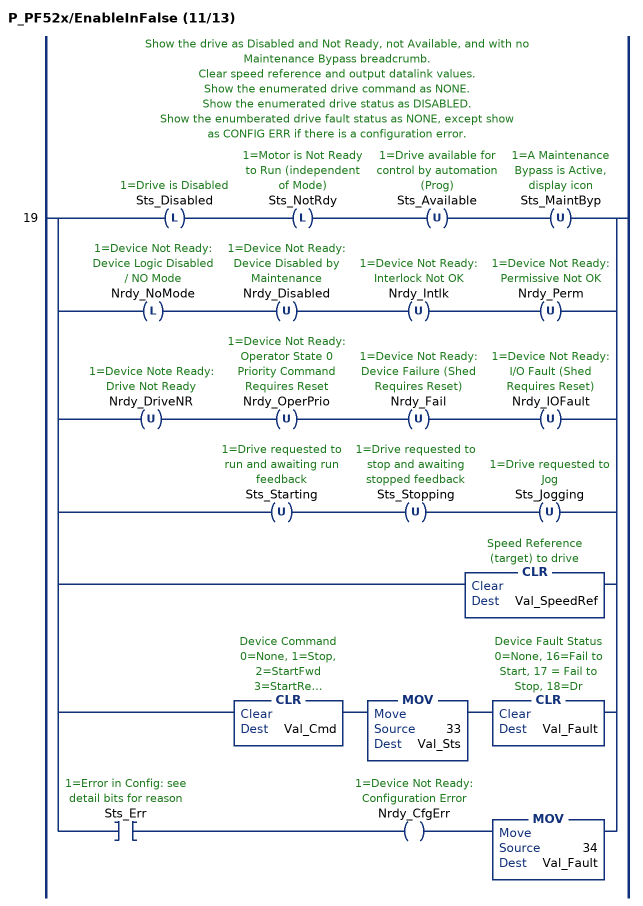
   // Show the drive as Disabled and Not Ready, not Available, and with no
   // Maintenance Bypass breadcrumb.
   // Clear speed reference and output datalink values.
   // Show the enumerated drive command as NONE.
   // Show the enumerated drive status as DISABLED.
   // Show the enumberated drive fault status as NONE, except show
   // as CONFIG ERR if there is a configuration error.
   19: [OTL(Sts_Disabled) OTL(Sts_NotRdy) OTU(Sts_Available) OTU(Sts_MaintByp) ,OTL(Nrdy_NoMode) OTU(Nrdy_Disabled) OTU(Nrdy_Intlk) OTU(Nrdy_Perm) ,OTU(Nrdy_DriveNR) OTU(Nrdy_OperPrio) OTU(Nrdy_Fail) OTU(Nrdy_IOFault) ,OTU(Sts_Starting) OTU(Sts_Stopping) OTU(Sts_Jogging) ,CLR(Val_SpeedRef) ,CLR(Val_Cmd) MOV(33,Val_Sts) CLR(Val_Fault) ,XIC(Sts_Err) OTE(Nrdy_CfgErr) MOV(34,Val_Fault) ];
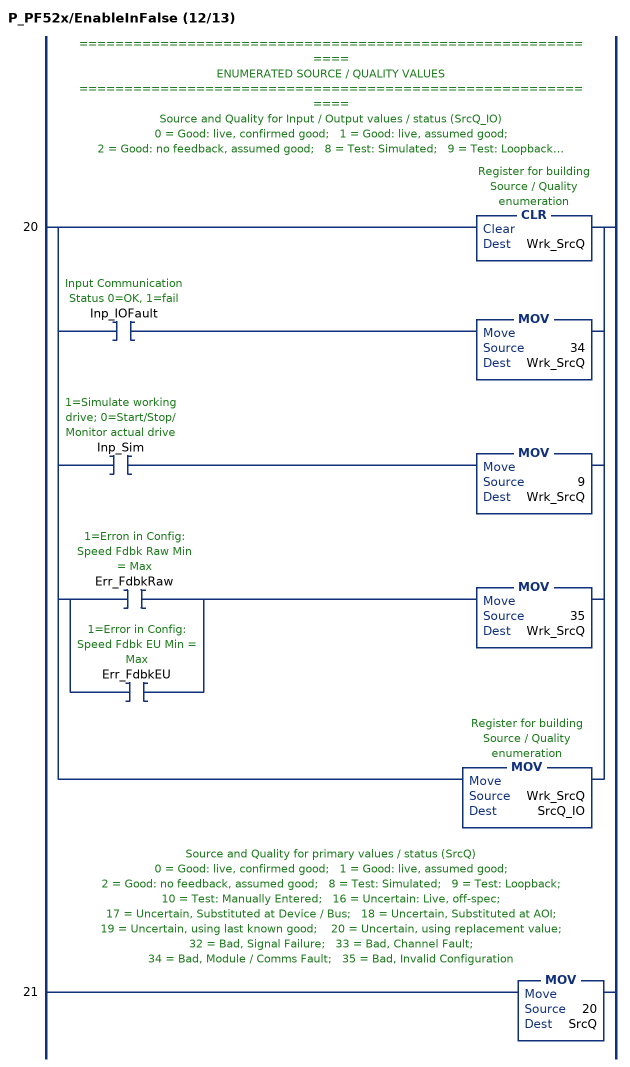
   // ============================================================
   // ENUMERATED SOURCE / QUALITY VALUES
   // ============================================================
   // Source and Quality for Input / Output values / status (SrcQ_IO)
   // 0 = Good: live, confirmed good;   1 = Good: live, assumed good;
   // 2 = Good: no feedback, assumed good;   8 = Test: Simulated;   9 = Test: Loopback;
   // 10 = Test: Manually Entered;   16 = Uncertain: Live, off-spec;
   // 17 = Uncertain, Substituted at Device / Bus;   18 = Uncertain, Substituted at AOI;
   // 19 = Uncertain, using last known good;    20 = Uncertain, using replacement value;
   // 32 = Bad, Signal Failure;   33 = Bad, Channel Fault;
   // 34 = Bad, Module / Comms Fault;   35 = Bad, Invalid Configuration
   20: [CLR(Wrk_SrcQ) ,XIC(Inp_IOFault) MOV(34,Wrk_SrcQ) ,XIC(Inp_Sim) MOV(9,Wrk_SrcQ) ,[XIC(Err_FdbkRaw) ,XIC(Err_FdbkEU) ] MOV(35,Wrk_SrcQ) ,MOV(Wrk_SrcQ,SrcQ_IO) ];
   // Source and Quality for primary values / status (SrcQ)
   // 0 = Good: live, confirmed good;   1 = Good: live, assumed good;
   // 2 = Good: no feedback, assumed good;   8 = Test: Simulated;   9 = Test: Loopback;
   // 10 = Test: Manually Entered;   16 = Uncertain: Live, off-spec;
   // 17 = Uncertain, Substituted at Device / Bus;   18 = Uncertain, Substituted at AOI;
   // 19 = Uncertain, using last known good;    20 = Uncertain, using replacement value;
   // 32 = Bad, Signal Failure;   33 = Bad, Channel Fault;
   // 34 = Bad, Module / Comms Fault;   35 = Bad, Invalid Configuration
   21: MOV(20,SrcQ);
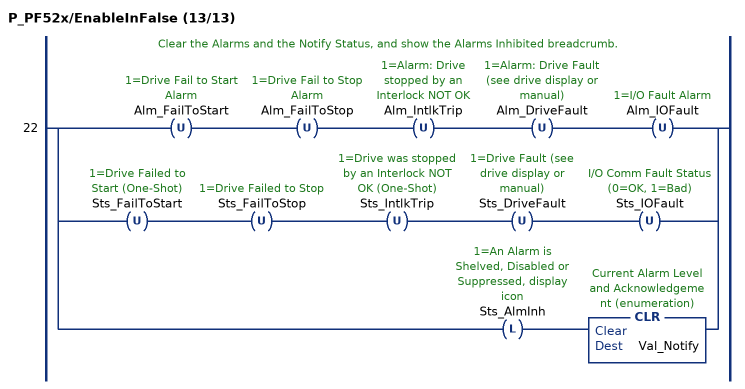
   // Clear the Alarms and the Notify Status, and show the Alarms Inhibited breadcrumb.
   22: [OTU(Alm_FailToStart) OTU(Alm_FailToStop) OTU(Alm_IntlkTrip) OTU(Alm_DriveFault) OTU(Alm_IOFault) ,OTU(Sts_FailToStart) OTU(Sts_FailToStop) OTU(Sts_IntlkTrip) OTU(Sts_DriveFault) OTU(Sts_IOFault) ,OTL(Sts_AlmInh) CLR(Val_Notify) ];
END_ROUTINE
